KUKA KRL program: EPS_2_26115_SA7012_A_20260219035554.src

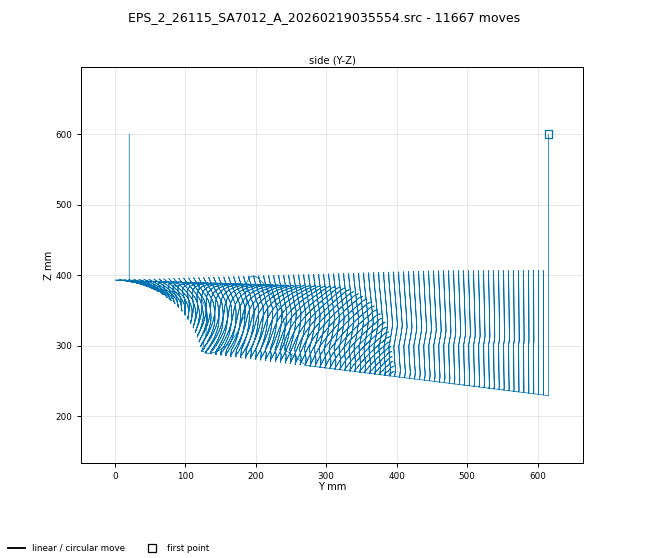
[picture p0: tool path of EPS_2_26115_SA7012_A_20260219035554.src, 11667 of 11669 moves have a stored position in this frame; points joined in program order, loops and branches not executed]
&ACCESS RVP
&REL 4
&COMMENT QRS 19112012
&PARAM EDITMASK = *
DEF PART()
EXT BAS (BAS_COMMAND :IN,REAL :IN )
INT I
BAS (#INITMOV,0 )

;KUKA QRS Post kuka4.cps  Date:22-06-2017 !

File_ID=3068

QRS_PRE_INIT()

;Init var - Until changes are made in qrs_pre_init
Outlet_Square_prg=0
Inlet_1_Square_prg=0
Inlet_2_Square_prg=0
Inlet_3_Square_prg=0
Inlet_4_Square_prg=0
Inlet_5_Square_prg=0

Outlet_1={X 0.000, Y 460.000, Z 306.500, B 0.000, E1 0.000 }
Inlet_1={X 0.000, Y 560.070, Z 281.500, B 0.000, E1 180.000 }
Outlet_1_type=201
Inlet_1_type=0
;QRS#1=Sidecore dimensions
;QRS#2=200-8" PVC SDR 35 Cut Back
;QRS#3=DeadEnd 201
;QRS#4=
;QRS#5=
;QRS#6=
;QRS#7=
;QRS#8=
;QRS#9=12-08 PSX
;QRS#10=

;QRS#11=
;QRS#12=
;QRS#13=
;QRS#14=
;QRS#15=
;QRS#16=1220x127x686 2,25'
;QRS#17=EPS Height
;QRS#18=407
;QRS#19=*
;QRS#20= UPDATED VERSION 22-06-2017
;QRS#21=*
Outlet_Square=0100
Inlet_1_Square=00
Inlet_2_Square=0
Inlet_3_Square=0
Inlet_4_Square=0
Inlet_5_Square=0
Mill_Square=1
Outlet_Square_Prg=214
Inlet_1_Square_prg=0

QRS_INIT()

$ADVANCE=5

; T1
PTP {E1 173.647,E2 173.647}
PTP {X 0,Y 615.427,A -85,B 0,C 180,E1 173.647,E2 173.647,E3 0,E4 0,E5 0,E6 0}
QRS_SPEED_INIT()
LIN {X 0,Y 615.427,Z 600,A -85,B 0,C 180,E1 173.647,E2 173.647,E3 0,E4 0,E5 0,E6 0} C_VEL
LIN {X 0,Y 615.427,Z 239.376,A -85,B 0,C 180,E1 173.647,E2 173.647} C_VEL
LIN {X 0,Y 615.427,Z 231.196,A -85,B 0,C 180,E1 173.647,E2 173.647} C_VEL
LIN {X 0,Y 615.428,Z 229.196,A -85,B 0,C 180,E1 173.461,E2 173.461} C_VEL
LIN {X 0,Y 615.493,Z 229.194,A -85,B 0,C 180,E1 170.806,E2 170.806} C_VEL
LIN {X 0,Y 615.44,Z 229.198,A -85,B 0,C 180,E1 168.143,E2 168.143} C_VEL
LIN {X 0,Y 615.432,Z 229.198,A -85,B 0,C 180,E1 166.084,E2 166.084} C_VEL
LIN {X 0,Y 615.43,Z 229.198,A -85,B 0,C 180,E1 164.098,E2 164.098} C_VEL
LIN {X 0,Y 615.426,Z 229.198,A -85,B 0,C 180,E1 162.046,E2 162.046} C_VEL
LIN {X 0,Y 615.472,Z 229.195,A -85,B 0,C 180,E1 159.274,E2 159.274} C_VEL
LIN {X 0,Y 615.435,Z 229.198,A -85,B 0,C 180,E1 156.447,E2 156.447} C_VEL
LIN {X 0,Y 615.425,Z 229.198,A -85,B 0,C 180,E1 154.287,E2 154.287} C_VEL
LIN {X 0,Y 615.424,Z 229.197,A -85,B 0,C 180,E1 152.088,E2 152.088} C_VEL
LIN {X 0,Y 615.437,Z 229.197,A -85,B 0,C 180,E1 149.844,E2 149.844} C_VEL
LIN {X 0,Y 615.473,Z 229.197,A -85,B 0,C 180,E1 147.548,E2 147.548} C_VEL
LIN {X 0,Y 615.476,Z 229.2,A -85,B 0,C 180,E1 145.191,E2 145.191} C_VEL
LIN {X 0,Y 615.429,Z 229.199,A -85,B 0,C 180,E1 142.761,E2 142.761} C_VEL
LIN {X 0,Y 615.456,Z 229.197,A -85,B 0,C 180,E1 139.913,E2 139.913} C_VEL
LIN {X 0,Y 615.499,Z 229.197,A -85,B 0,C 180,E1 137.656,E2 137.656} C_VEL
LIN {X 0,Y 615.424,Z 229.199,A -85,B 0,C 180,E1 134.934,E2 134.934} C_VEL
LIN {X 0,Y 615.463,Z 229.197,A -85,B 0,C 180,E1 132.087,E2 132.087} C_VEL
LIN {X 0,Y 615.485,Z 229.201,A -85,B 0,C 180,E1 129.749,E2 129.749} C_VEL
LIN {X 0,Y 615.428,Z 229.199,A -85,B 0,C 180,E1 127.246,E2 127.246} C_VEL
LIN {X 0,Y 615.421,Z 229.198,A -85,B 0,C 180,E1 124.819,E2 124.819} C_VEL
LIN {X 0,Y 615.465,Z 229.198,A -85,B 0,C 180,E1 122.34,E2 122.34} C_VEL
LIN {X 0,Y 615.456,Z 229.2,A -85,B 0,C 180,E1 119.803,E2 119.803} C_VEL
LIN {X 0,Y 615.416,Z 229.199,A -85,B 0,C 180,E1 117.18,E2 117.18} C_VEL
LIN {X 0,Y 615.483,Z 229.204,A -85,B 0,C 180,E1 114.272,E2 114.272} C_VEL
LIN {X 0,Y 615.466,Z 229.201,A -85,B 0,C 180,E1 112.137,E2 112.137} C_VEL
LIN {X 0,Y 615.449,Z 229.2,A -85,B 0,C 180,E1 110.034,E2 110.034} C_VEL
LIN {X 0,Y 615.435,Z 229.2,A -85,B 0,C 180,E1 107.958,E2 107.958} C_VEL
LIN {X 0,Y 615.427,Z 229.2,A -85,B 0,C 180,E1 105.906,E2 105.906} C_VEL
LIN {X 0,Y 615.421,Z 229.2,A -85,B 0,C 180,E1 103.875,E2 103.875} C_VEL
LIN {X 0,Y 615.418,Z 229.2,A -85,B 0,C 180,E1 101.862,E2 101.862} C_VEL
LIN {X 0,Y 615.416,Z 229.2,A -85,B 0,C 180,E1 99.863,E2 99.863} C_VEL
LIN {X 0,Y 615.413,Z 229.2,A -85,B 0,C 180,E1 97.876,E2 97.876} C_VEL
LIN {X 0,Y 615.413,Z 229.2,A -85,B 0,C 180,E1 95.899,E2 95.899} C_VEL
LIN {X 0,Y 615.448,Z 229.2,A -85,B 0,C 180,E1 93.273,E2 93.273} C_VEL
LIN {X 0,Y 615.453,Z 229.2,A -85,B 0,C 180,E1 90.654,E2 90.654} C_VEL
LIN {X 0,Y 615.413,Z 229.2,A -85,B 0,C 180,E1 88.037,E2 88.037} C_VEL
LIN {X 0,Y 615.459,Z 229.2,A -85,B 0,C 180,E1 85.415,E2 85.415} C_VEL
LIN {X 0,Y 615.44,Z 229.2,A -85,B 0,C 180,E1 82.784,E2 82.784} C_VEL
LIN {X 0,Y 615.439,Z 229.199,A -85,B 0,C 180,E1 80.801,E2 80.801} C_VEL
LIN {X 0,Y 615.435,Z 229.199,A -85,B 0,C 180,E1 78.806,E2 78.806} C_VEL
LIN {X 0,Y 615.43,Z 229.199,A -85,B 0,C 180,E1 76.798,E2 76.798} C_VEL
LIN {X 0,Y 615.425,Z 229.199,A -85,B 0,C 180,E1 74.773,E2 74.773} C_VEL
LIN {X 0,Y 615.42,Z 229.199,A -85,B 0,C 180,E1 72.728,E2 72.728} C_VEL
LIN {X 0,Y 615.417,Z 229.199,A -85,B 0,C 180,E1 70.66,E2 70.66} C_VEL
LIN {X 0,Y 615.416,Z 229.199,A -85,B 0,C 180,E1 68.566,E2 68.566} C_VEL
LIN {X 0,Y 615.461,Z 229.2,A -85,B 0,C 180,E1 65.98,E2 65.98} C_VEL
LIN {X 0,Y 615.471,Z 229.198,A -85,B 0,C 180,E1 63.556,E2 63.556} C_VEL
LIN {X 0,Y 615.441,Z 229.198,A -85,B 0,C 180,E1 61.34,E2 61.34} C_VEL
LIN {X 0,Y 615.42,Z 229.199,A -85,B 0,C 180,E1 59.077,E2 59.077} C_VEL
LIN {X 0,Y 615.441,Z 229.199,A -85,B 0,C 180,E1 56.46,E2 56.46} C_VEL
LIN {X 0,Y 615.443,Z 229.198,A -85,B 0,C 180,E1 53.573,E2 53.573} C_VEL
LIN {X 0,Y 615.422,Z 229.199,A -85,B 0,C 180,E1 50.935,E2 50.935} C_VEL
LIN {X 0,Y 615.459,Z 229.2,A -85,B 0,C 180,E1 48.525,E2 48.525} C_VEL
LIN {X 0,Y 615.446,Z 229.198,A -85,B 0,C 180,E1 45.848,E2 45.848} C_VEL
LIN {X 0,Y 615.421,Z 229.198,A -85,B 0,C 180,E1 43.242,E2 43.242} C_VEL
LIN {X 0,Y 615.428,Z 229.199,A -85,B 0,C 180,E1 41.089,E2 41.089} C_VEL
LIN {X 0,Y 615.45,Z 229.199,A -85,B 0,C 180,E1 38.899,E2 38.899} C_VEL
LIN {X 0,Y 615.473,Z 229.2,A -85,B 0,C 180,E1 36.418,E2 36.418} C_VEL
LIN {X 0,Y 615.437,Z 229.197,A -85,B 0,C 180,E1 34.018,E2 34.018} C_VEL
LIN {X 0,Y 615.42,Z 229.198,A -85,B 0,C 180,E1 31.683,E2 31.683} C_VEL
LIN {X 0,Y 615.433,Z 229.199,A -85,B 0,C 180,E1 29.403,E2 29.403} C_VEL
LIN {X 0,Y 615.476,Z 229.2,A -85,B 0,C 180,E1 27.045,E2 27.045} C_VEL
LIN {X 0,Y 615.436,Z 229.197,A -85,B 0,C 180,E1 24.268,E2 24.268} C_VEL
LIN {X 0,Y 615.427,Z 229.197,A -85,B 0,C 180,E1 22.133,E2 22.133} C_VEL
LIN {X 0,Y 615.424,Z 229.197,A -85,B 0,C 180,E1 20.03,E2 20.03} C_VEL
LIN {X 0,Y 615.481,Z 229.201,A -85,B 0,C 180,E1 17.266,E2 17.266} C_VEL
LIN {X 0,Y 615.436,Z 229.196,A -85,B 0,C 180,E1 14.545,E2 14.545} C_VEL
LIN {X 0,Y 615.433,Z 229.196,A -85,B 0,C 180,E1 12.527,E2 12.527} C_VEL
LIN {X 0,Y 615.431,Z 229.196,A -85,B 0,C 180,E1 10.523,E2 10.523} C_VEL
LIN {X 0,Y 615.428,Z 229.197,A -85,B 0,C 180,E1 8.533,E2 8.533} C_VEL
LIN {X 0,Y 615.428,Z 229.196,A -85,B 0,C 180,E1 6.539,E2 6.539} C_VEL
LIN {X 0,Y 615.428,Z 229.196,A -85,B 0,C 180,E1 4.581,E2 4.581} C_VEL
LIN {X 0,Y 615.457,Z 229.199,A -85,B 0,C 180,E1 1.959,E2 1.959} C_VEL
LIN {X 0,Y 615.473,Z 229.194,A -85,B 0,C 180,E1 -0.658,E2 -0.658} C_VEL
LIN {X 0,Y 615.428,Z 229.196,A -85,B 0,C 180,E1 -3.277,E2 -3.277} C_VEL
LIN {X 0,Y 615.467,Z 229.199,A -85,B 0,C 180,E1 -5.902,E2 -5.902} C_VEL
LIN {X 0,Y 615.463,Z 229.194,A -85,B 0,C 180,E1 -8.54,E2 -8.54} C_VEL
LIN {X 0,Y 615.43,Z 229.197,A -85,B 0,C 180,E1 -11.197,E2 -11.197} C_VEL
LIN {X 0,Y 615.499,Z 229.199,A -85,B 0,C 180,E1 -13.941,E2 -13.941} C_VEL
LIN {X 0,Y 615.438,Z 229.195,A -85,B 0,C 180,E1 -16.591,E2 -16.591} C_VEL
LIN {X 0,Y 615.435,Z 229.195,A -85,B 0,C 180,E1 -18.65,E2 -18.65} C_VEL
LIN {X 0,Y 615.432,Z 229.196,A -85,B 0,C 180,E1 -20.735,E2 -20.735} C_VEL
LIN {X 0,Y 615.481,Z 229.202,A -85,B 0,C 180,E1 -23.559,E2 -23.559} C_VEL
LIN {X 0,Y 615.499,Z 229.194,A -85,B 0,C 180,E1 -25.718,E2 -25.718} C_VEL
LIN {X 0,Y 615.43,Z 229.197,A -85,B 0,C 180,E1 -28.663,E2 -28.663} C_VEL
LIN {X 0,Y 615.462,Z 229.199,A -85,B 0,C 180,E1 -31.084,E2 -31.084} C_VEL
LIN {X 0,Y 615.447,Z 229.194,A -85,B 0,C 180,E1 -34.027,E2 -34.027} C_VEL
LIN {X 0,Y 615.434,Z 229.196,A -85,B 0,C 180,E1 -36.431,E2 -36.431} C_VEL
LIN {X 0,Y 615.488,Z 229.2,A -85,B 0,C 180,E1 -39.063,E2 -39.063} C_VEL
LIN {X 0,Y 615.482,Z 229.191,A -85,B 0,C 180,E1 -41.476,E2 -41.476} C_VEL
LIN {X 0,Y 615.435,Z 229.195,A -85,B 0,C 180,E1 -44.156,E2 -44.156} C_VEL
LIN {X 0,Y 615.478,Z 229.199,A -85,B 0,C 180,E1 -46.756,E2 -46.756} C_VEL
LIN {X 0,Y 615.478,Z 229.338,A -85,B 0,C 180,E1 -48.716,E2 -48.716} C_VEL
LIN {X 0,Y 615.493,Z 234.318,A -85,B 0,C 180,E1 -51.097,E2 -51.097} C_VEL
LIN {X 0,Y 615.453,Z 239.696,A -85,B 0,C 180,E1 -53.574,E2 -53.574} C_VEL
LIN {X 0,Y 615.494,Z 246.171,A -85,B 0,C 180,E1 -56.467,E2 -56.467} C_VEL
LIN {X 0,Y 615.478,Z 252.224,A -85,B 0,C 180,E1 -59.08,E2 -59.08} C_VEL
LIN {X 0,Y 615.475,Z 258.104,A -85,B 0,C 180,E1 -61.553,E2 -61.553} C_VEL
LIN {X 0,Y 615.479,Z 264.742,A -85,B 0,C 180,E1 -64.284,E2 -64.284} C_VEL
LIN {X 0,Y 615.484,Z 270.106,A -85,B 0,C 180,E1 -66.444,E2 -66.444} C_VEL
LIN {X 0,Y 615.489,Z 277.253,A -85,B 0,C 180,E1 -69.27,E2 -69.27} C_VEL
LIN {X 0,Y 615.465,Z 284.402,A -85,B 0,C 180,E1 -72.043,E2 -72.043} C_VEL
LIN {X 0,Y 615.495,Z 291.538,A -85,B 0,C 180,E1 -74.774,E2 -74.774} C_VEL
LIN {X 0,Y 615.442,Z 298.683,A -85,B 0,C 180,E1 -77.469,E2 -77.469} C_VEL
LIN {X 0,Y 615.497,Z 301.074,A -85,B 0,C 180,E1 -78.369,E2 -78.369} C_VEL
LIN {X 0,Y 615.482,Z 316.869,A -85,B 0,C 180,E1 -78.724,E2 -78.724} C_VEL
LIN {X 0,Y 615.443,Z 329.251,A -85,B 0,C 180,E1 -79.136,E2 -79.136} C_VEL
LIN {X 0,Y 615.439,Z 340.489,A -85,B 0,C 180,E1 -79.639,E2 -79.639} C_VEL
LIN {X 0,Y 615.489,Z 351.997,A -85,B 0,C 180,E1 -80.304,E2 -80.304} C_VEL
LIN {X 0,Y 615.499,Z 362.343,A -85,B 0,C 180,E1 -81.05,E2 -81.05} C_VEL
LIN {X 0,Y 615.497,Z 370.813,A -85,B 0,C 180,E1 -81.794,E2 -81.794} C_VEL
LIN {X 0,Y 615.498,Z 378.607,A -85,B 0,C 180,E1 -82.62,E2 -82.62} C_VEL
LIN {X 0,Y 615.496,Z 386.204,A -85,B 0,C 180,E1 -83.608,E2 -83.608} C_VEL
LIN {X 0,Y 615.498,Z 393.205,A -85,B 0,C 180,E1 -84.759,E2 -84.759} C_VEL
LIN {X 0,Y 615.493,Z 397.852,A -85,B 0,C 180,E1 -85.744,E2 -85.744} C_VEL
LIN {X 0,Y 615.494,Z 401.399,A -85,B 0,C 180,E1 -86.727,E2 -86.727} C_VEL
LIN {X 0,Y 615.497,Z 403.233,A -85,B 0,C 180,E1 -87.382,E2 -87.382} C_VEL
LIN {X 0,Y 615.5,Z 404.608,A -85,B 0,C 180,E1 -88.037,E2 -88.037} C_VEL
LIN {X 0,Y 615.496,Z 406.173,A -85,B 0,C 180,E1 -89.346,E2 -89.346} C_VEL
LIN {X 0,Y 615.494,Z 406.389,A -85,B 0,C 180,E1 -90,E2 -90} C_VEL
LIN {X 0,Y 615.495,Z 405.58,A -85,B 0,C 180,E1 -91.309,E2 -91.309} C_VEL
LIN {X 0,Y 615.5,Z 404.608,A -85,B 0,C 180,E1 -91.963,E2 -91.963} C_VEL
LIN {X 0,Y 615.497,Z 403.233,A -85,B 0,C 180,E1 -92.618,E2 -92.618} C_VEL
LIN {X 0,Y 615.496,Z 400.35,A -85,B 0,C 180,E1 -93.601,E2 -93.601} C_VEL
LIN {X 0,Y 615.498,Z 396.442,A -85,B 0,C 180,E1 -94.584,E2 -94.584} C_VEL
LIN {X 0,Y 615.499,Z 391.405,A -85,B 0,C 180,E1 -95.57,E2 -95.57} C_VEL
LIN {X 0,Y 615.497,Z 384.875,A -85,B 0,C 180,E1 -96.583,E2 -96.583} C_VEL
LIN {X 0,Y 615.497,Z 377.134,A -85,B 0,C 180,E1 -97.545,E2 -97.545} C_VEL
LIN {X 0,Y 615.498,Z 369.047,A -85,B 0,C 180,E1 -98.371,E2 -98.371} C_VEL
LIN {X 0,Y 615.499,Z 359.17,A -85,B 0,C 180,E1 -99.198,E2 -99.198} C_VEL
LIN {X 0,Y 615.471,Z 347.987,A -85,B 0,C 180,E1 -99.945,E2 -99.945} C_VEL
LIN {X 0,Y 615.435,Z 337.035,A -85,B 0,C 180,E1 -100.528,E2 -100.528} C_VEL
LIN {X 0,Y 615.454,Z 324.825,A -85,B 0,C 180,E1 -101.029,E2 -101.029} C_VEL
LIN {X 0,Y 615.495,Z 312.073,A -85,B 0,C 180,E1 -101.401,E2 -101.401} C_VEL
LIN {X 0,Y 615.497,Z 301.074,A -85,B 0,C 180,E1 -101.631,E2 -101.631} C_VEL
LIN {X 0,Y 615.467,Z 294.99,A -85,B 0,C 180,E1 -103.923,E2 -103.923} C_VEL
LIN {X 0,Y 615.463,Z 287.97,A -85,B 0,C 180,E1 -106.587,E2 -106.587} C_VEL
LIN {X 0,Y 615.487,Z 280.835,A -85,B 0,C 180,E1 -109.338,E2 -109.338} C_VEL
LIN {X 0,Y 615.474,Z 273.68,A -85,B 0,C 180,E1 -112.137,E2 -112.137} C_VEL
LIN {X 0,Y 615.483,Z 266.537,A -85,B 0,C 180,E1 -114.991,E2 -114.991} C_VEL
LIN {X 0,Y 615.489,Z 259.377,A -85,B 0,C 180,E1 -117.914,E2 -117.914} C_VEL
LIN {X 0,Y 615.48,Z 254.015,A -85,B 0,C 180,E1 -120.16,E2 -120.16} C_VEL
LIN {X 0,Y 615.461,Z 248.65,A -85,B 0,C 180,E1 -122.458,E2 -122.458} C_VEL
LIN {X 0,Y 615.476,Z 243.274,A -85,B 0,C 180,E1 -124.815,E2 -124.815} C_VEL
LIN {X 0,Y 615.491,Z 237.901,A -85,B 0,C 180,E1 -127.241,E2 -127.241} C_VEL
LIN {X 0,Y 615.443,Z 232.534,A -85,B 0,C 180,E1 -129.753,E2 -129.753} C_VEL
LIN {X 0,Y 615.469,Z 229.199,A -85,B 0,C 180,E1 -131.379,E2 -131.379} C_VEL
LIN {X 0,Y 615.436,Z 229.195,A -85,B 0,C 180,E1 -133.991,E2 -133.991} C_VEL
LIN {X 0,Y 615.437,Z 229.195,A -85,B 0,C 180,E1 -136.006,E2 -136.006} C_VEL
LIN {X 0,Y 615.478,Z 229.192,A -85,B 0,C 180,E1 -138.523,E2 -138.523} C_VEL
LIN {X 0,Y 615.468,Z 229.199,A -85,B 0,C 180,E1 -141.092,E2 -141.092} C_VEL
LIN {X 0,Y 615.434,Z 229.196,A -85,B 0,C 180,E1 -143.569,E2 -143.569} C_VEL
LIN {X 0,Y 615.496,Z 229.193,A -85,B 0,C 180,E1 -146.463,E2 -146.463} C_VEL
LIN {X 0,Y 615.447,Z 229.198,A -85,B 0,C 180,E1 -149.076,E2 -149.076} C_VEL
LIN {X 0,Y 615.432,Z 229.196,A -85,B 0,C 180,E1 -151.557,E2 -151.557} C_VEL
LIN {X 0,Y 615.5,Z 229.199,A -85,B 0,C 180,E1 -154.427,E2 -154.427} C_VEL
LIN {X 0,Y 615.432,Z 229.196,A -85,B 0,C 180,E1 -157.151,E2 -157.151} C_VEL
LIN {X 0,Y 615.479,Z 229.194,A -85,B 0,C 180,E1 -159.964,E2 -159.964} C_VEL
LIN {X 0,Y 615.441,Z 229.198,A -85,B 0,C 180,E1 -162.725,E2 -162.725} C_VEL
LIN {X 0,Y 615.436,Z 229.197,A -85,B 0,C 180,E1 -164.77,E2 -164.77} C_VEL
LIN {X 0,Y 615.433,Z 229.197,A -85,B 0,C 180,E1 -166.794,E2 -166.794} C_VEL
LIN {X 0,Y 615.434,Z 229.195,A -85,B 0,C 180,E1 -169.132,E2 -169.132} C_VEL
LIN {X 0,Y 615.463,Z 229.194,A -85,B 0,C 180,E1 -171.46,E2 -171.46} C_VEL
LIN {X 0,Y 615.467,Z 229.199,A -85,B 0,C 180,E1 -174.098,E2 -174.098} C_VEL
LIN {X 0,Y 615.428,Z 229.196,A -85,B 0,C 180,E1 -176.723,E2 -176.723} C_VEL
LIN {X 0,Y 615.47,Z 229.195,A -85,B 0,C 180,E1 -179.342,E2 -179.342} C_VEL
LIN {X 0,Y 615.457,Z 229.199,A -85,B 0,C 180,E1 -181.959,E2 -181.959} C_VEL
LIN {X 0,Y 615.428,Z 229.196,A -85,B 0,C 180,E1 -184.581,E2 -184.581} C_VEL
LIN {X 0,Y 615.428,Z 229.196,A -85,B 0,C 180,E1 -186.539,E2 -186.539} C_VEL
LIN {X 0,Y 614.793,Z 229.344,A -85,B 0,C 180,E1 -187.085,E2 -187.085} C_VEL
LIN {X 0,Y 611.998,Z 229.748,A -85,B 0,C 180,E1 -187.971,E2 -187.971} C_VEL
LIN {X 0,Y 609.607,Z 230.064,A -85,B 0,C 180,E1 -188.684,E2 -188.684} C_VEL
LIN {X 0,Y 608.552,Z 230.185,A -85,B 0,C 180,E1 -189.234,E2 -189.234} C_VEL
LIN {X 0,Y 608.451,Z 230.194,A -85,B 0,C 180,E1 -189.42,E2 -189.42} C_VEL
LIN {X 0,Y 608.418,Z 230.193,A -85,B 0,C 180,E1 -191.996,E2 -191.996} C_VEL
LIN {X 0,Y 608.399,Z 230.195,A -85,B 0,C 180,E1 -194.034,E2 -194.034} C_VEL
LIN {X 0,Y 608.429,Z 230.192,A -85,B 0,C 180,E1 -196.52,E2 -196.52} C_VEL
LIN {X 0,Y 608.419,Z 230.195,A -85,B 0,C 180,E1 -199.566,E2 -199.566} C_VEL
LIN {X 0,Y 608.429,Z 230.192,A -85,B 0,C 180,E1 -202.401,E2 -202.401} C_VEL
LIN {X 0,Y 608.421,Z 230.196,A -85,B 0,C 180,E1 -205.296,E2 -205.296} C_VEL
LIN {X 0,Y 608.408,Z 230.194,A -85,B 0,C 180,E1 -207.514,E2 -207.514} C_VEL
LIN {X 0,Y 608.411,Z 230.193,A -85,B 0,C 180,E1 -209.964,E2 -209.964} C_VEL
LIN {X 0,Y 608.423,Z 230.199,A -85,B 0,C 180,E1 -212.875,E2 -212.875} C_VEL
LIN {X 0,Y 608.401,Z 230.195,A -85,B 0,C 180,E1 -215.273,E2 -215.273} C_VEL
LIN {X 0,Y 608.423,Z 230.192,A -85,B 0,C 180,E1 -217.742,E2 -217.742} C_VEL
LIN {X 0,Y 608.435,Z 230.198,A -85,B 0,C 180,E1 -220.328,E2 -220.328} C_VEL
LIN {X 0,Y 608.404,Z 230.196,A -85,B 0,C 180,E1 -222.956,E2 -222.956} C_VEL
LIN {X 0,Y 608.396,Z 230.195,A -85,B 0,C 180,E1 -225.2,E2 -225.2} C_VEL
LIN {X 0,Y 608.44,Z 230.194,A -85,B 0,C 180,E1 -227.938,E2 -227.938} C_VEL
LIN {X 0,Y 608.426,Z 230.193,A -85,B 0,C 180,E1 -230.697,E2 -230.697} C_VEL
LIN {X 0,Y 608.39,Z 230.195,A -85,B 0,C 180,E1 -233.081,E2 -233.081} C_VEL
LIN {X 0,Y 608.428,Z 230.193,A -85,B 0,C 180,E1 -235.529,E2 -235.529} C_VEL
LIN {X 0,Y 608.437,Z 230.199,A -85,B 0,C 180,E1 -237.905,E2 -237.905} C_VEL
LIN {X 0,Y 608.438,Z 230.194,A -85,B 0,C 180,E1 -240.219,E2 -240.219} C_VEL
LIN {X 0,Y 608.411,Z 230.193,A -85,B 0,C 180,E1 -242.79,E2 -242.79} C_VEL
LIN {X 0,Y 608.453,Z 230.196,A -85,B 0,C 180,E1 -245.836,E2 -245.836} C_VEL
LIN {X 0,Y 608.417,Z 230.193,A -85,B 0,C 180,E1 -248.307,E2 -248.307} C_VEL
LIN {X 0,Y 608.431,Z 230.194,A -85,B 0,C 180,E1 -251.13,E2 -251.13} C_VEL
LIN {X 0,Y 608.417,Z 230.196,A -85,B 0,C 180,E1 -253.905,E2 -253.905} C_VEL
LIN {X 0,Y 608.402,Z 230.196,A -85,B 0,C 180,E1 -255.978,E2 -255.978} C_VEL
LIN {X 0,Y 608.406,Z 230.195,A -85,B 0,C 180,E1 -257.999,E2 -257.999} C_VEL
LIN {X 0,Y 608.395,Z 230.196,A -85,B 0,C 180,E1 -260.022,E2 -260.022} C_VEL
LIN {X 0,Y 608.411,Z 230.193,A -85,B 0,C 180,E1 -262.032,E2 -262.032} C_VEL
LIN {X 0,Y 608.42,Z 230.195,A -85,B 0,C 180,E1 -264.698,E2 -264.698} C_VEL
LIN {X 0,Y 608.442,Z 230.195,A -85,B 0,C 180,E1 -267.352,E2 -267.352} C_VEL
LIN {X 0,Y 608.403,Z 230.194,A -85,B 0,C 180,E1 -270,E2 -270} C_VEL
LIN {X 0,Y 608.442,Z 230.195,A -85,B 0,C 180,E1 -272.648,E2 -272.648} C_VEL
LIN {X 0,Y 608.42,Z 230.195,A -85,B 0,C 180,E1 -275.302,E2 -275.302} C_VEL
LIN {X 0,Y 608.411,Z 230.193,A -85,B 0,C 180,E1 -277.968,E2 -277.968} C_VEL
LIN {X 0,Y 608.444,Z 230.199,A -85,B 0,C 180,E1 -280.65,E2 -280.65} C_VEL
LIN {X 0,Y 608.405,Z 230.194,A -85,B 0,C 180,E1 -283.357,E2 -283.357} C_VEL
LIN {X 0,Y 608.409,Z 230.193,A -85,B 0,C 180,E1 -285.407,E2 -285.407} C_VEL
LIN {X 0,Y 608.39,Z 230.195,A -85,B 0,C 180,E1 -287.478,E2 -287.478} C_VEL
LIN {X 0,Y 608.393,Z 230.195,A -85,B 0,C 180,E1 -289.572,E2 -289.572} C_VEL
LIN {X 0,Y 608.476,Z 230.194,A -85,B 0,C 180,E1 -292.405,E2 -292.405} C_VEL
LIN {X 0,Y 608.418,Z 230.197,A -85,B 0,C 180,E1 -294.572,E2 -294.572} C_VEL
LIN {X 0,Y 608.411,Z 230.193,A -85,B 0,C 180,E1 -297.21,E2 -297.21} C_VEL
LIN {X 0,Y 608.468,Z 230.194,A -85,B 0,C 180,E1 -299.985,E2 -299.985} C_VEL
LIN {X 0,Y 608.404,Z 230.194,A -85,B 0,C 180,E1 -302.882,E2 -302.882} C_VEL
LIN {X 0,Y 608.397,Z 230.196,A -85,B 0,C 180,E1 -305.28,E2 -305.28} C_VEL
LIN {X 0,Y 608.438,Z 230.194,A -85,B 0,C 180,E1 -308.247,E2 -308.247} C_VEL
LIN {X 0,Y 608.426,Z 230.193,A -85,B 0,C 180,E1 -310.336,E2 -310.336} C_VEL
LIN {X 0,Y 608.395,Z 230.195,A -85,B 0,C 180,E1 -312.964,E2 -312.964} C_VEL
LIN {X 0,Y 608.439,Z 230.198,A -85,B 0,C 180,E1 -315.737,E2 -315.737} C_VEL
LIN {X 0,Y 608.437,Z 230.194,A -85,B 0,C 180,E1 -317.945,E2 -317.945} C_VEL
LIN {X 0,Y 608.395,Z 230.195,A -85,B 0,C 180,E1 -320.71,E2 -320.71} C_VEL
LIN {X 0,Y 608.424,Z 230.196,A -85,B 0,C 180,E1 -323.09,E2 -323.09} C_VEL
LIN {X 0,Y 608.452,Z 230.195,A -85,B 0,C 180,E1 -325.537,E2 -325.537} C_VEL
LIN {X 0,Y 608.425,Z 230.192,A -85,B 0,C 180,E1 -327.91,E2 -327.91} C_VEL
LIN {X 0,Y 608.409,Z 230.193,A -85,B 0,C 180,E1 -330.224,E2 -330.224} C_VEL
LIN {X 0,Y 608.454,Z 230.192,A -85,B 0,C 180,E1 -332.795,E2 -332.795} C_VEL
LIN {X 0,Y 608.425,Z 230.191,A -85,B 0,C 180,E1 -335.856,E2 -335.856} C_VEL
LIN {X 0,Y 608.425,Z 230.192,A -85,B 0,C 180,E1 -338.312,E2 -338.312} C_VEL
LIN {X 0,Y 608.441,Z 230.193,A -85,B 0,C 180,E1 -341.289,E2 -341.289} C_VEL
LIN {X 0,Y 608.408,Z 230.193,A -85,B 0,C 180,E1 -343.91,E2 -343.91} C_VEL
LIN {X 0,Y 608.458,Z 230.197,A -85,B 0,C 180,E1 -346.648,E2 -346.648} C_VEL
LIN {X 0,Y 608.42,Z 230.192,A -85,B 0,C 180,E1 -349.354,E2 -349.354} C_VEL
LIN {X 0,Y 608.412,Z 230.193,A -85,B 0,C 180,E1 -351.368,E2 -351.368} C_VEL
LIN {X 0,Y 608.424,Z 230.194,A -85,B 0,C 180,E1 -354.037,E2 -354.037} C_VEL
LIN {X 0,Y 608.467,Z 230.191,A -85,B 0,C 180,E1 -356.693,E2 -356.693} C_VEL
LIN {X 0,Y 608.407,Z 230.193,A -85,B 0,C 180,E1 -359.342,E2 -359.342} C_VEL
LIN {X 0,Y 608.416,Z 230.192,A -85,B 0,C 180,E1 -361.328,E2 -361.328} C_VEL
LIN {X 0,Y 608.4,Z 230.194,A -85,B 0,C 180,E1 -363.315,E2 -363.315} C_VEL
LIN {X 0,Y 608.442,Z 230.197,A -85,B 0,C 180,E1 -365.971,E2 -365.971} C_VEL
LIN {X 0,Y 608.43,Z 230.192,A -85,B 0,C 180,E1 -368.64,E2 -368.64} C_VEL
LIN {X 0,Y 608.414,Z 230.194,A -85,B 0,C 180,E1 -371.328,E2 -371.328} C_VEL
LIN {X 0,Y 608.468,Z 230.194,A -85,B 0,C 180,E1 -374.041,E2 -374.041} C_VEL
LIN {X 0,Y 608.412,Z 230.193,A -85,B 0,C 180,E1 -376.788,E2 -376.788} C_VEL
LIN {X 0,Y 608.431,Z 230.198,A -85,B 0,C 180,E1 -379.574,E2 -379.574} C_VEL
LIN {X 0,Y 608.43,Z 230.191,A -85,B 0,C 180,E1 -382.472,E2 -382.472} C_VEL
LIN {X 0,Y 608.418,Z 230.192,A -85,B 0,C 180,E1 -384.575,E2 -384.575} C_VEL
LIN {X 0,Y 608.405,Z 230.194,A -85,B 0,C 180,E1 -386.779,E2 -386.779} C_VEL
LIN {X 0,Y 608.465,Z 230.191,A -85,B 0,C 180,E1 -389.782,E2 -389.782} C_VEL
LIN {X 0,Y 608.416,Z 230.192,A -85,B 0,C 180,E1 -392.517,E2 -392.517} C_VEL
LIN {X 0,Y 608.418,Z 230.196,A -85,B 0,C 180,E1 -394.903,E2 -394.903} C_VEL
LIN {X 0,Y 608.445,Z 230.191,A -85,B 0,C 180,E1 -397.75,E2 -397.75} C_VEL
LIN {X 0,Y 608.406,Z 230.194,A -85,B 0,C 180,E1 -400.325,E2 -400.325} C_VEL
LIN {X 0,Y 608.449,Z 230.198,A -85,B 0,C 180,E1 -402.962,E2 -402.962} C_VEL
LIN {X 0,Y 608.42,Z 230.193,A -85,B 0,C 180,E1 -405.742,E2 -405.742} C_VEL
LIN {X 0,Y 608.455,Z 230.313,A -85,B 0,C 180,E1 -408.525,E2 -408.525} C_VEL
LIN {X 0,Y 608.474,Z 234.678,A -85,B 0,C 180,E1 -410.704,E2 -410.704} C_VEL
LIN {X 0,Y 608.473,Z 239.769,A -85,B 0,C 180,E1 -413.087,E2 -413.087} C_VEL
LIN {X 0,Y 608.453,Z 245.159,A -85,B 0,C 180,E1 -415.53,E2 -415.53} C_VEL
LIN {X 0,Y 608.454,Z 250.548,A -85,B 0,C 180,E1 -417.906,E2 -417.906} C_VEL
LIN {X 0,Y 608.476,Z 255.938,A -85,B 0,C 180,E1 -420.222,E2 -420.222} C_VEL
LIN {X 0,Y 608.459,Z 262.086,A -85,B 0,C 180,E1 -422.798,E2 -422.798} C_VEL
LIN {X 0,Y 608.454,Z 268.513,A -85,B 0,C 180,E1 -425.429,E2 -425.429} C_VEL
LIN {X 0,Y 608.445,Z 275.699,A -85,B 0,C 180,E1 -428.308,E2 -428.308} C_VEL
LIN {X 0,Y 608.432,Z 282.885,A -85,B 0,C 180,E1 -431.13,E2 -431.13} C_VEL
LIN {X 0,Y 608.422,Z 290.071,A -85,B 0,C 180,E1 -433.905,E2 -433.905} C_VEL
LIN {X 0,Y 608.429,Z 297.257,A -85,B 0,C 180,E1 -436.643,E2 -436.643} C_VEL
LIN {X 0,Y 608.459,Z 301.63,A -85,B 0,C 180,E1 -438.254,E2 -438.254} C_VEL
LIN {X 0,Y 608.544,Z 314.708,A -85,B 0,C 180,E1 -438.53,E2 -438.53} C_VEL
LIN {X 0,Y 608.473,Z 327.572,A -85,B 0,C 180,E1 -438.942,E2 -438.942} C_VEL
LIN {X 0,Y 608.465,Z 338.926,A -85,B 0,C 180,E1 -439.435,E2 -439.435} C_VEL
LIN {X 0,Y 608.471,Z 349.581,A -85,B 0,C 180,E1 -440.023,E2 -440.023} C_VEL
LIN {X 0,Y 608.483,Z 360.477,A -85,B 0,C 180,E1 -440.778,E2 -440.778} C_VEL
LIN {X 0,Y 608.475,Z 371.114,A -85,B 0,C 180,E1 -441.699,E2 -441.699} C_VEL
LIN {X 0,Y 608.471,Z 378.961,A -85,B 0,C 180,E1 -442.534,E2 -442.534} C_VEL
LIN {X 0,Y 608.461,Z 386.29,A -85,B 0,C 180,E1 -443.485,E2 -443.485} C_VEL
LIN {X 0,Y 608.451,Z 391.866,A -85,B 0,C 180,E1 -444.366,E2 -444.366} C_VEL
LIN {X 0,Y 608.432,Z 396.951,A -85,B 0,C 180,E1 -445.362,E2 -445.362} C_VEL
LIN {X 0,Y 608.449,Z 400.896,A -85,B 0,C 180,E1 -446.358,E2 -446.358} C_VEL
LIN {X 0,Y 608.425,Z 403.809,A -85,B 0,C 180,E1 -447.352,E2 -447.352} C_VEL
LIN {X 0,Y 608.445,Z 405.201,A -85,B 0,C 180,E1 -448.014,E2 -448.014} C_VEL
LIN {X 0,Y 608.439,Z 406.783,A -85,B 0,C 180,E1 -449.338,E2 -449.338} C_VEL
LIN {X 0,Y 608.434,Z 406.999,A -85,B 0,C 180,E1 -450,E2 -450} C_VEL
LIN {X 0,Y 608.448,Z 406.184,A -85,B 0,C 180,E1 -451.324,E2 -451.324} C_VEL
LIN {X 0,Y 608.445,Z 405.201,A -85,B 0,C 180,E1 -451.986,E2 -451.986} C_VEL
LIN {X 0,Y 608.425,Z 403.809,A -85,B 0,C 180,E1 -452.648,E2 -452.648} C_VEL
LIN {X 0,Y 608.449,Z 400.896,A -85,B 0,C 180,E1 -453.642,E2 -453.642} C_VEL
LIN {X 0,Y 608.432,Z 396.951,A -85,B 0,C 180,E1 -454.638,E2 -454.638} C_VEL
LIN {X 0,Y 608.438,Z 390.877,A -85,B 0,C 180,E1 -455.801,E2 -455.801} C_VEL
LIN {X 0,Y 608.463,Z 384.236,A -85,B 0,C 180,E1 -456.799,E2 -456.799} C_VEL
LIN {X 0,Y 608.456,Z 375.991,A -85,B 0,C 180,E1 -457.8,E2 -457.8} C_VEL
LIN {X 0,Y 608.472,Z 367.535,A -85,B 0,C 180,E1 -458.636,E2 -458.636} C_VEL
LIN {X 0,Y 608.48,Z 357.091,A -85,B 0,C 180,E1 -459.473,E2 -459.473} C_VEL
LIN {X 0,Y 608.481,Z 346.758,A -85,B 0,C 180,E1 -460.145,E2 -460.145} C_VEL
LIN {X 0,Y 608.46,Z 335.898,A -85,B 0,C 180,E1 -460.711,E2 -460.711} C_VEL
LIN {X 0,Y 608.49,Z 324.113,A -85,B 0,C 180,E1 -461.185,E2 -461.185} C_VEL
LIN {X 0,Y 608.55,Z 311.273,A -85,B 0,C 180,E1 -461.554,E2 -461.554} C_VEL
LIN {X 0,Y 608.435,Z 301.468,A -85,B 0,C 180,E1 -461.768,E2 -461.768} C_VEL
LIN {X 0,Y 608.426,Z 295.461,A -85,B 0,C 180,E1 -464.038,E2 -464.038} C_VEL
LIN {X 0,Y 608.42,Z 288.275,A -85,B 0,C 180,E1 -466.785,E2 -466.785} C_VEL
LIN {X 0,Y 608.447,Z 281.089,A -85,B 0,C 180,E1 -469.57,E2 -469.57} C_VEL
LIN {X 0,Y 608.445,Z 275.699,A -85,B 0,C 180,E1 -471.692,E2 -471.692} C_VEL
LIN {X 0,Y 608.454,Z 268.513,A -85,B 0,C 180,E1 -474.571,E2 -474.571} C_VEL
LIN {X 0,Y 608.459,Z 262.086,A -85,B 0,C 180,E1 -477.202,E2 -477.202} C_VEL
LIN {X 0,Y 608.469,Z 255.487,A -85,B 0,C 180,E1 -479.97,E2 -479.97} C_VEL
LIN {X 0,Y 608.442,Z 249.579,A -85,B 0,C 180,E1 -482.518,E2 -482.518} C_VEL
LIN {X 0,Y 608.471,Z 244.18,A -85,B 0,C 180,E1 -484.907,E2 -484.907} C_VEL
LIN {X 0,Y 608.444,Z 237.973,A -85,B 0,C 180,E1 -487.747,E2 -487.747} C_VEL
LIN {X 0,Y 608.44,Z 232.537,A -85,B 0,C 180,E1 -490.326,E2 -490.326} C_VEL
LIN {X 0,Y 608.455,Z 230.318,A -85,B 0,C 180,E1 -491.475,E2 -491.475} C_VEL
LIN {X 0,Y 608.431,Z 230.191,A -85,B 0,C 180,E1 -493.872,E2 -493.872} C_VEL
LIN {X 0,Y 608.482,Z 230.19,A -85,B 0,C 180,E1 -496.689,E2 -496.689} C_VEL
LIN {X 0,Y 608.454,Z 230.197,A -85,B 0,C 180,E1 -498.821,E2 -498.821} C_VEL
LIN {X 0,Y 608.413,Z 230.195,A -85,B 0,C 180,E1 -501.406,E2 -501.406} C_VEL
LIN {X 0,Y 608.435,Z 230.19,A -85,B 0,C 180,E1 -503.955,E2 -503.955} C_VEL
LIN {X 0,Y 608.449,Z 230.192,A -85,B 0,C 180,E1 -506.326,E2 -506.326} C_VEL
LIN {X 0,Y 608.442,Z 230.198,A -85,B 0,C 180,E1 -508.732,E2 -508.732} C_VEL
LIN {X 0,Y 608.427,Z 230.191,A -85,B 0,C 180,E1 -511.386,E2 -511.386} C_VEL
LIN {X 0,Y 608.483,Z 230.191,A -85,B 0,C 180,E1 -514.275,E2 -514.275} C_VEL
LIN {X 0,Y 608.421,Z 230.194,A -85,B 0,C 180,E1 -516.872,E2 -516.872} C_VEL
LIN {X 0,Y 608.428,Z 230.191,A -85,B 0,C 180,E1 -519.328,E2 -519.328} C_VEL
LIN {X 0,Y 608.438,Z 230.193,A -85,B 0,C 180,E1 -521.825,E2 -521.825} C_VEL
LIN {X 0,Y 608.439,Z 230.193,A -85,B 0,C 180,E1 -524.59,E2 -524.59} C_VEL
LIN {X 0,Y 608.427,Z 230.193,A -85,B 0,C 180,E1 -526.64,E2 -526.64} C_VEL
LIN {X 0,Y 608.429,Z 230.192,A -85,B 0,C 180,E1 -529.346,E2 -529.346} C_VEL
LIN {X 0,Y 608.464,Z 230.195,A -85,B 0,C 180,E1 -532.029,E2 -532.029} C_VEL
LIN {X 0,Y 608.414,Z 230.193,A -85,B 0,C 180,E1 -534.694,E2 -534.694} C_VEL
LIN {X 0,Y 608.462,Z 230.19,A -85,B 0,C 180,E1 -537.348,E2 -537.348} C_VEL
LIN {X 0,Y 608.452,Z 230.193,A -85,B 0,C 180,E1 -539.996,E2 -539.996} C_VEL
LIN {X 0,Y 608.425,Z 230.191,A -85,B 0,C 180,E1 -542.644,E2 -542.644} C_VEL
LIN {X 0,Y 608.459,Z 230.193,A -85,B 0,C 180,E1 -545.298,E2 -545.298} C_VEL
LIN {X 0,Y 608.409,Z 230.196,A -85,B 0,C 180,E1 -547.963,E2 -547.963} C_VEL
LIN {X 0,Y 608.451,Z 230.194,A -85,B 0,C 180,E1 -549.42,E2 -549.42} C_VEL
LIN {X 0,Y 607.745,Z 230.278,A -85,B 0,C 180,E1 -549.972,E2 -549.972} C_VEL
LIN {X 0,Y 604.876,Z 230.636,A -85,B 0,C 180,E1 -550.869,E2 -550.869} C_VEL
LIN {X 0,Y 602.479,Z 230.938,A -85,B 0,C 180,E1 -551.591,E2 -551.591} C_VEL
LIN {X 0,Y 601.455,Z 231.06,A -85,B 0,C 180,E1 -552.147,E2 -552.147} C_VEL
LIN {X 0,Y 601.373,Z 231.07,A -85,B 0,C 180,E1 -552.336,E2 -552.336} C_VEL
LIN {X 0,Y 601.385,Z 231.073,A -85,B 0,C 180,E1 -554.893,E2 -554.893} C_VEL
LIN {X 0,Y 601.391,Z 231.074,A -85,B 0,C 180,E1 -556.982,E2 -556.982} C_VEL
LIN {X 0,Y 601.37,Z 231.071,A -85,B 0,C 180,E1 -559.805,E2 -559.805} C_VEL
LIN {X 0,Y 601.387,Z 231.072,A -85,B 0,C 180,E1 -562.601,E2 -562.601} C_VEL
LIN {X 0,Y 601.374,Z 231.079,A -85,B 0,C 180,E1 -564.874,E2 -564.874} C_VEL
LIN {X 0,Y 601.383,Z 231.071,A -85,B 0,C 180,E1 -567.358,E2 -567.358} C_VEL
LIN {X 0,Y 601.376,Z 231.071,A -85,B 0,C 180,E1 -569.389,E2 -569.389} C_VEL
LIN {X 0,Y 601.362,Z 231.071,A -85,B 0,C 180,E1 -571.723,E2 -571.723} C_VEL
LIN {X 0,Y 601.388,Z 231.07,A -85,B 0,C 180,E1 -574.114,E2 -574.114} C_VEL
LIN {X 0,Y 601.377,Z 231.079,A -85,B 0,C 180,E1 -576.577,E2 -576.577} C_VEL
LIN {X 0,Y 601.366,Z 231.072,A -85,B 0,C 180,E1 -579.122,E2 -579.122} C_VEL
LIN {X 0,Y 601.382,Z 231.07,A -85,B 0,C 180,E1 -581.76,E2 -581.76} C_VEL
LIN {X 0,Y 601.373,Z 231.077,A -85,B 0,C 180,E1 -584.531,E2 -584.531} C_VEL
LIN {X 0,Y 601.358,Z 231.071,A -85,B 0,C 180,E1 -587.326,E2 -587.326} C_VEL
LIN {X 0,Y 601.372,Z 231.077,A -85,B 0,C 180,E1 -590.003,E2 -590.003} C_VEL
LIN {X 0,Y 601.38,Z 231.071,A -85,B 0,C 180,E1 -592.614,E2 -592.614} C_VEL
LIN {X 0,Y 601.374,Z 231.069,A -85,B 0,C 180,E1 -595.066,E2 -595.066} C_VEL
LIN {X 0,Y 601.388,Z 231.07,A -85,B 0,C 180,E1 -597.482,E2 -597.482} C_VEL
LIN {X 0,Y 601.434,Z 231.071,A -85,B 0,C 180,E1 -599.837,E2 -599.837} C_VEL
LIN {X 0,Y 601.388,Z 231.068,A -85,B 0,C 180,E1 -602.886,E2 -602.886} C_VEL
LIN {X 0,Y 601.428,Z 231.071,A -85,B 0,C 180,E1 -605.859,E2 -605.859} C_VEL
LIN {X 0,Y 601.383,Z 231.072,A -85,B 0,C 180,E1 -608.04,E2 -608.04} C_VEL
LIN {X 0,Y 601.357,Z 231.073,A -85,B 0,C 180,E1 -610.189,E2 -610.189} C_VEL
LIN {X 0,Y 601.38,Z 231.072,A -85,B 0,C 180,E1 -613.013,E2 -613.013} C_VEL
LIN {X 0,Y 601.356,Z 231.075,A -85,B 0,C 180,E1 -615.903,E2 -615.903} C_VEL
LIN {X 0,Y 601.367,Z 231.073,A -85,B 0,C 180,E1 -617.857,E2 -617.857} C_VEL
LIN {X 0,Y 601.363,Z 231.072,A -85,B 0,C 180,E1 -620.583,E2 -620.583} C_VEL
LIN {X 0,Y 601.422,Z 231.073,A -85,B 0,C 180,E1 -623.289,E2 -623.289} C_VEL
LIN {X 0,Y 601.34,Z 231.074,A -85,B 0,C 180,E1 -625.979,E2 -625.979} C_VEL
LIN {X 0,Y 601.355,Z 231.072,A -85,B 0,C 180,E1 -627.991,E2 -627.991} C_VEL
LIN {X 0,Y 601.41,Z 231.07,A -85,B 0,C 180,E1 -630.67,E2 -630.67} C_VEL
LIN {X 0,Y 601.386,Z 231.072,A -85,B 0,C 180,E1 -633.35,E2 -633.35} C_VEL
LIN {X 0,Y 601.349,Z 231.073,A -85,B 0,C 180,E1 -636.038,E2 -636.038} C_VEL
LIN {X 0,Y 601.415,Z 231.075,A -85,B 0,C 180,E1 -638.738,E2 -638.738} C_VEL
LIN {X 0,Y 601.372,Z 231.07,A -85,B 0,C 180,E1 -641.459,E2 -641.459} C_VEL
LIN {X 0,Y 601.355,Z 231.072,A -85,B 0,C 180,E1 -643.517,E2 -643.517} C_VEL
LIN {X 0,Y 601.409,Z 231.072,A -85,B 0,C 180,E1 -646.287,E2 -646.287} C_VEL
LIN {X 0,Y 601.373,Z 231.071,A -85,B 0,C 180,E1 -649.1,E2 -649.1} C_VEL
LIN {X 0,Y 601.353,Z 231.072,A -85,B 0,C 180,E1 -651.241,E2 -651.241} C_VEL
LIN {X 0,Y 601.369,Z 231.07,A -85,B 0,C 180,E1 -653.412,E2 -653.412} C_VEL
LIN {X 0,Y 601.366,Z 231.075,A -85,B 0,C 180,E1 -655.874,E2 -655.874} C_VEL
LIN {X 0,Y 601.391,Z 231.07,A -85,B 0,C 180,E1 -658.628,E2 -658.628} C_VEL
LIN {X 0,Y 601.38,Z 231.069,A -85,B 0,C 180,E1 -660.944,E2 -660.944} C_VEL
LIN {X 0,Y 601.384,Z 231.069,A -85,B 0,C 180,E1 -663.316,E2 -663.316} C_VEL
LIN {X 0,Y 601.393,Z 231.072,A -85,B 0,C 180,E1 -666.271,E2 -666.271} C_VEL
LIN {X 0,Y 601.385,Z 231.069,A -85,B 0,C 180,E1 -669.128,E2 -669.128} C_VEL
LIN {X 0,Y 601.387,Z 231.078,A -85,B 0,C 180,E1 -671.767,E2 -671.767} C_VEL
LIN {X 0,Y 601.372,Z 231.07,A -85,B 0,C 180,E1 -674.539,E2 -674.539} C_VEL
LIN {X 0,Y 601.412,Z 231.072,A -85,B 0,C 180,E1 -677.408,E2 -677.408} C_VEL
LIN {X 0,Y 601.366,Z 231.07,A -85,B 0,C 180,E1 -680.472,E2 -680.472} C_VEL
LIN {X 0,Y 601.391,Z 231.068,A -85,B 0,C 180,E1 -682.622,E2 -682.622} C_VEL
LIN {X 0,Y 601.412,Z 231.07,A -85,B 0,C 180,E1 -685.075,E2 -685.075} C_VEL
LIN {X 0,Y 601.411,Z 231.072,A -85,B 0,C 180,E1 -687.49,E2 -687.49} C_VEL
LIN {X 0,Y 601.389,Z 231.069,A -85,B 0,C 180,E1 -689.856,E2 -689.856} C_VEL
LIN {X 0,Y 601.366,Z 231.07,A -85,B 0,C 180,E1 -692.136,E2 -692.136} C_VEL
LIN {X 0,Y 601.385,Z 231.069,A -85,B 0,C 180,E1 -694.386,E2 -694.386} C_VEL
LIN {X 0,Y 601.384,Z 231.072,A -85,B 0,C 180,E1 -696.594,E2 -696.594} C_VEL
LIN {X 0,Y 601.396,Z 231.069,A -85,B 0,C 180,E1 -699.482,E2 -699.482} C_VEL
LIN {X 0,Y 601.366,Z 231.073,A -85,B 0,C 180,E1 -702.316,E2 -702.316} C_VEL
LIN {X 0,Y 601.391,Z 231.072,A -85,B 0,C 180,E1 -704.413,E2 -704.413} C_VEL
LIN {X 0,Y 601.391,Z 231.07,A -85,B 0,C 180,E1 -707.176,E2 -707.176} C_VEL
LIN {X 0,Y 601.391,Z 231.069,A -85,B 0,C 180,E1 -709.228,E2 -709.228} C_VEL
LIN {X 0,Y 601.383,Z 231.07,A -85,B 0,C 180,E1 -711.943,E2 -711.943} C_VEL
LIN {X 0,Y 601.419,Z 231.071,A -85,B 0,C 180,E1 -714.64,E2 -714.64} C_VEL
LIN {X 0,Y 601.396,Z 231.067,A -85,B 0,C 180,E1 -717.325,E2 -717.325} C_VEL
LIN {X 0,Y 601.421,Z 231.069,A -85,B 0,C 180,E1 -720.004,E2 -720.004} C_VEL
LIN {X 0,Y 601.425,Z 231.066,A -85,B 0,C 180,E1 -722.683,E2 -722.683} C_VEL
LIN {X 0,Y 601.383,Z 231.069,A -85,B 0,C 180,E1 -725.368,E2 -725.368} C_VEL
LIN {X 0,Y 601.427,Z 231.073,A -85,B 0,C 180,E1 -728.064,E2 -728.064} C_VEL
LIN {X 0,Y 601.383,Z 231.068,A -85,B 0,C 180,E1 -730.997,E2 -730.997} C_VEL
LIN {X 0,Y 601.392,Z 231.071,A -85,B 0,C 180,E1 -733.52,E2 -733.52} C_VEL
LIN {X 0,Y 601.408,Z 231.068,A -85,B 0,C 180,E1 -736.291,E2 -736.291} C_VEL
LIN {X 0,Y 601.399,Z 231.068,A -85,B 0,C 180,E1 -739.102,E2 -739.102} C_VEL
LIN {X 0,Y 601.389,Z 231.073,A -85,B 0,C 180,E1 -741.963,E2 -741.963} C_VEL
LIN {X 0,Y 601.379,Z 231.07,A -85,B 0,C 180,E1 -744.882,E2 -744.882} C_VEL
LIN {X 0,Y 601.398,Z 231.074,A -85,B 0,C 180,E1 -747.361,E2 -747.361} C_VEL
LIN {X 0,Y 601.401,Z 231.067,A -85,B 0,C 180,E1 -750.168,E2 -750.168} C_VEL
LIN {X 0,Y 601.391,Z 231.069,A -85,B 0,C 180,E1 -752.712,E2 -752.712} C_VEL
LIN {X 0,Y 601.377,Z 231.077,A -85,B 0,C 180,E1 -755.111,E2 -755.111} C_VEL
LIN {X 0,Y 601.433,Z 231.069,A -85,B 0,C 180,E1 -757.421,E2 -757.421} C_VEL
LIN {X 0,Y 601.38,Z 231.069,A -85,B 0,C 180,E1 -760,E2 -760} C_VEL
LIN {X 0,Y 601.376,Z 231.074,A -85,B 0,C 180,E1 -762.675,E2 -762.675} C_VEL
LIN {X 0,Y 601.403,Z 231.07,A -85,B 0,C 180,E1 -765.481,E2 -765.481} C_VEL
LIN {X 0,Y 601.407,Z 231.182,A -85,B 0,C 180,E1 -768.234,E2 -768.234} C_VEL
LIN {X 0,Y 601.452,Z 234.38,A -85,B 0,C 180,E1 -770.009,E2 -770.009} C_VEL
LIN {X 0,Y 601.443,Z 239.847,A -85,B 0,C 180,E1 -772.619,E2 -772.619} C_VEL
LIN {X 0,Y 601.444,Z 245.159,A -85,B 0,C 180,E1 -775.071,E2 -775.071} C_VEL
LIN {X 0,Y 601.413,Z 250.548,A -85,B 0,C 180,E1 -777.484,E2 -777.484} C_VEL
LIN {X 0,Y 601.434,Z 255.974,A -85,B 0,C 180,E1 -779.852,E2 -779.852} C_VEL
LIN {X 0,Y 601.404,Z 262.537,A -85,B 0,C 180,E1 -782.641,E2 -782.641} C_VEL
LIN {X 0,Y 601.398,Z 268.513,A -85,B 0,C 180,E1 -785.122,E2 -785.122} C_VEL
LIN {X 0,Y 601.378,Z 274.123,A -85,B 0,C 180,E1 -787.405,E2 -787.405} C_VEL
LIN {X 0,Y 601.372,Z 281.089,A -85,B 0,C 180,E1 -790.19,E2 -790.19} C_VEL
LIN {X 0,Y 601.342,Z 288.275,A -85,B 0,C 180,E1 -793.012,E2 -793.012} C_VEL
LIN {X 0,Y 601.352,Z 295.835,A -85,B 0,C 180,E1 -795.937,E2 -795.937} C_VEL
LIN {X 0,Y 601.368,Z 301.624,A -85,B 0,C 180,E1 -798.113,E2 -798.113} C_VEL
LIN {X 0,Y 601.591,Z 312.182,A -85,B 0,C 180,E1 -798.332,E2 -798.332} C_VEL
LIN {X 0,Y 601.53,Z 324.409,A -85,B 0,C 180,E1 -798.694,E2 -798.694} C_VEL
LIN {X 0,Y 601.454,Z 337.179,A -85,B 0,C 180,E1 -799.225,E2 -799.225} C_VEL
LIN {X 0,Y 601.46,Z 348.17,A -85,B 0,C 180,E1 -799.821,E2 -799.821} C_VEL
LIN {X 0,Y 601.455,Z 359.396,A -85,B 0,C 180,E1 -800.585,E2 -800.585} C_VEL
LIN {X 0,Y 601.423,Z 369.34,A -85,B 0,C 180,E1 -801.432,E2 -801.432} C_VEL
LIN {X 0,Y 601.418,Z 378.959,A -85,B 0,C 180,E1 -802.446,E2 -802.446} C_VEL
LIN {X 0,Y 601.371,Z 386.226,A -85,B 0,C 180,E1 -803.399,E2 -803.399} C_VEL
LIN {X 0,Y 601.372,Z 391.863,A -85,B 0,C 180,E1 -804.299,E2 -804.299} C_VEL
LIN {X 0,Y 601.336,Z 396.951,A -85,B 0,C 180,E1 -805.307,E2 -805.307} C_VEL
LIN {X 0,Y 601.368,Z 400.896,A -85,B 0,C 180,E1 -806.315,E2 -806.315} C_VEL
LIN {X 0,Y 601.325,Z 403.807,A -85,B 0,C 180,E1 -807.32,E2 -807.32} C_VEL
LIN {X 0,Y 601.343,Z 405.2,A -85,B 0,C 180,E1 -807.991,E2 -807.991} C_VEL
LIN {X 0,Y 601.339,Z 406.783,A -85,B 0,C 180,E1 -809.33,E2 -809.33} C_VEL
LIN {X 0,Y 601.335,Z 406.995,A -85,B 0,C 180,E1 -810,E2 -810} C_VEL
LIN {X 0,Y 601.348,Z 406.185,A -85,B 0,C 180,E1 -811.339,E2 -811.339} C_VEL
LIN {X 0,Y 601.343,Z 405.2,A -85,B 0,C 180,E1 -812.009,E2 -812.009} C_VEL
LIN {X 0,Y 601.325,Z 403.807,A -85,B 0,C 180,E1 -812.68,E2 -812.68} C_VEL
LIN {X 0,Y 601.368,Z 400.896,A -85,B 0,C 180,E1 -813.685,E2 -813.685} C_VEL
LIN {X 0,Y 601.336,Z 396.951,A -85,B 0,C 180,E1 -814.693,E2 -814.693} C_VEL
LIN {X 0,Y 601.372,Z 391.863,A -85,B 0,C 180,E1 -815.701,E2 -815.701} C_VEL
LIN {X 0,Y 601.383,Z 385.472,A -85,B 0,C 180,E1 -816.711,E2 -816.711} C_VEL
LIN {X 0,Y 601.396,Z 377.481,A -85,B 0,C 180,E1 -817.723,E2 -817.723} C_VEL
LIN {X 0,Y 601.423,Z 369.34,A -85,B 0,C 180,E1 -818.568,E2 -818.568} C_VEL
LIN {X 0,Y 601.455,Z 359.396,A -85,B 0,C 180,E1 -819.415,E2 -819.415} C_VEL
LIN {X 0,Y 601.46,Z 348.17,A -85,B 0,C 180,E1 -820.179,E2 -820.179} C_VEL
LIN {X 0,Y 601.454,Z 337.179,A -85,B 0,C 180,E1 -820.775,E2 -820.775} C_VEL
LIN {X 0,Y 601.532,Z 324.774,A -85,B 0,C 180,E1 -821.293,E2 -821.293} C_VEL
LIN {X 0,Y 601.591,Z 312.182,A -85,B 0,C 180,E1 -821.668,E2 -821.668} C_VEL
LIN {X 0,Y 601.368,Z 301.624,A -85,B 0,C 180,E1 -821.887,E2 -821.887} C_VEL
LIN {X 0,Y 601.338,Z 293.664,A -85,B 0,C 180,E1 -824.899,E2 -824.899} C_VEL
LIN {X 0,Y 601.356,Z 286.478,A -85,B 0,C 180,E1 -827.689,E2 -827.689} C_VEL
LIN {X 0,Y 601.366,Z 279.292,A -85,B 0,C 180,E1 -830.524,E2 -830.524} C_VEL
LIN {X 0,Y 601.388,Z 272.106,A -85,B 0,C 180,E1 -833.411,E2 -833.411} C_VEL
LIN {X 0,Y 601.397,Z 266.128,A -85,B 0,C 180,E1 -835.862,E2 -835.862} C_VEL
LIN {X 0,Y 601.423,Z 259.159,A -85,B 0,C 180,E1 -838.785,E2 -838.785} C_VEL
LIN {X 0,Y 601.444,Z 252.955,A -85,B 0,C 180,E1 -841.457,E2 -841.457} C_VEL
LIN {X 0,Y 601.425,Z 246.955,A -85,B 0,C 180,E1 -844.118,E2 -844.118} C_VEL
LIN {X 0,Y 601.439,Z 241.566,A -85,B 0,C 180,E1 -846.58,E2 -846.58} C_VEL
LIN {X 0,Y 601.445,Z 235.322,A -85,B 0,C 180,E1 -849.534,E2 -849.534} C_VEL
LIN {X 0,Y 601.451,Z 231.463,A -85,B 0,C 180,E1 -851.594,E2 -851.594} C_VEL
LIN {X 0,Y 601.407,Z 231.183,A -85,B 0,C 180,E1 -851.766,E2 -851.766} C_VEL
LIN {X 0,Y 601.402,Z 231.07,A -85,B 0,C 180,E1 -854.531,E2 -854.531} C_VEL
LIN {X 0,Y 601.376,Z 231.074,A -85,B 0,C 180,E1 -857.325,E2 -857.325} C_VEL
LIN {X 0,Y 601.38,Z 231.069,A -85,B 0,C 180,E1 -860,E2 -860} C_VEL
LIN {X 0,Y 601.436,Z 231.069,A -85,B 0,C 180,E1 -862.617,E2 -862.617} C_VEL
LIN {X 0,Y 601.384,Z 231.073,A -85,B 0,C 180,E1 -865.064,E2 -865.064} C_VEL
LIN {X 0,Y 601.389,Z 231.068,A -85,B 0,C 180,E1 -867.479,E2 -867.479} C_VEL
LIN {X 0,Y 601.402,Z 231.067,A -85,B 0,C 180,E1 -869.854,E2 -869.854} C_VEL
LIN {X 0,Y 601.407,Z 231.069,A -85,B 0,C 180,E1 -872.884,E2 -872.884} C_VEL
LIN {X 0,Y 601.379,Z 231.07,A -85,B 0,C 180,E1 -875.118,E2 -875.118} C_VEL
LIN {X 0,Y 601.389,Z 231.073,A -85,B 0,C 180,E1 -878.037,E2 -878.037} C_VEL
LIN {X 0,Y 601.399,Z 231.068,A -85,B 0,C 180,E1 -880.898,E2 -880.898} C_VEL
LIN {X 0,Y 601.408,Z 231.068,A -85,B 0,C 180,E1 -883.709,E2 -883.709} C_VEL
LIN {X 0,Y 601.392,Z 231.071,A -85,B 0,C 180,E1 -886.48,E2 -886.48} C_VEL
LIN {X 0,Y 601.371,Z 231.07,A -85,B 0,C 180,E1 -889.22,E2 -889.22} C_VEL
LIN {X 0,Y 601.427,Z 231.073,A -85,B 0,C 180,E1 -891.936,E2 -891.936} C_VEL
LIN {X 0,Y 601.383,Z 231.069,A -85,B 0,C 180,E1 -894.632,E2 -894.632} C_VEL
LIN {X 0,Y 601.425,Z 231.066,A -85,B 0,C 180,E1 -897.317,E2 -897.317} C_VEL
LIN {X 0,Y 601.421,Z 231.069,A -85,B 0,C 180,E1 -899.996,E2 -899.996} C_VEL
LIN {X 0,Y 601.396,Z 231.067,A -85,B 0,C 180,E1 -902.675,E2 -902.675} C_VEL
LIN {X 0,Y 601.419,Z 231.071,A -85,B 0,C 180,E1 -905.36,E2 -905.36} C_VEL
LIN {X 0,Y 601.383,Z 231.07,A -85,B 0,C 180,E1 -908.057,E2 -908.057} C_VEL
LIN {X 0,Y 601.443,Z 231.066,A -85,B 0,C 180,E1 -911.026,E2 -911.026} C_VEL
LIN {X 0,Y 601.373,Z 231.07,A -85,B 0,C 180,E1 -912.336,E2 -912.336} C_VEL
LIN {X 0,Y 600.711,Z 231.157,A -85,B 0,C 180,E1 -912.895,E2 -912.895} C_VEL
LIN {X 0,Y 597.861,Z 231.514,A -85,B 0,C 180,E1 -913.803,E2 -913.803} C_VEL
LIN {X 0,Y 595.45,Z 231.816,A -85,B 0,C 180,E1 -914.533,E2 -914.533} C_VEL
LIN {X 0,Y 594.413,Z 231.945,A -85,B 0,C 180,E1 -915.096,E2 -915.096} C_VEL
LIN {X 0,Y 594.327,Z 231.952,A -85,B 0,C 180,E1 -915.287,E2 -915.287} C_VEL
LIN {X 0,Y 594.316,Z 231.949,A -85,B 0,C 180,E1 -917.901,E2 -917.901} C_VEL
LIN {X 0,Y 594.376,Z 231.947,A -85,B 0,C 180,E1 -920.771,E2 -920.771} C_VEL
LIN {X 0,Y 594.348,Z 231.945,A -85,B 0,C 180,E1 -923.7,E2 -923.7} C_VEL
LIN {X 0,Y 594.355,Z 231.951,A -85,B 0,C 180,E1 -926.695,E2 -926.695} C_VEL
LIN {X 0,Y 594.35,Z 231.952,A -85,B 0,C 180,E1 -928.994,E2 -928.994} C_VEL
LIN {X 0,Y 594.338,Z 231.946,A -85,B 0,C 180,E1 -931.638,E2 -931.638} C_VEL
LIN {X 0,Y 594.362,Z 231.952,A -85,B 0,C 180,E1 -934.574,E2 -934.574} C_VEL
LIN {X 0,Y 594.344,Z 231.948,A -85,B 0,C 180,E1 -937.082,E2 -937.082} C_VEL
LIN {X 0,Y 594.318,Z 231.949,A -85,B 0,C 180,E1 -939.769,E2 -939.769} C_VEL
LIN {X 0,Y 594.355,Z 231.953,A -85,B 0,C 180,E1 -942.368,E2 -942.368} C_VEL
LIN {X 0,Y 594.311,Z 231.949,A -85,B 0,C 180,E1 -945.187,E2 -945.187} C_VEL
LIN {X 0,Y 594.343,Z 231.954,A -85,B 0,C 180,E1 -948.146,E2 -948.146} C_VEL
LIN {X 0,Y 594.336,Z 231.946,A -85,B 0,C 180,E1 -951.192,E2 -951.192} C_VEL
LIN {X 0,Y 594.346,Z 231.95,A -85,B 0,C 180,E1 -953.756,E2 -953.756} C_VEL
LIN {X 0,Y 594.338,Z 231.952,A -85,B 0,C 180,E1 -956.237,E2 -956.237} C_VEL
LIN {X 0,Y 594.334,Z 231.947,A -85,B 0,C 180,E1 -958.648,E2 -958.648} C_VEL
LIN {X 0,Y 594.336,Z 231.947,A -85,B 0,C 180,E1 -961.036,E2 -961.036} C_VEL
LIN {X 0,Y 594.339,Z 231.953,A -85,B 0,C 180,E1 -963.971,E2 -963.971} C_VEL
LIN {X 0,Y 594.346,Z 231.947,A -85,B 0,C 180,E1 -966.295,E2 -966.295} C_VEL
LIN {X 0,Y 594.365,Z 231.946,A -85,B 0,C 180,E1 -969.223,E2 -969.223} C_VEL
LIN {X 0,Y 594.327,Z 231.95,A -85,B 0,C 180,E1 -972.095,E2 -972.095} C_VEL
LIN {X 0,Y 594.318,Z 231.949,A -85,B 0,C 180,E1 -974.218,E2 -974.218} C_VEL
LIN {X 0,Y 594.35,Z 231.949,A -85,B 0,C 180,E1 -977.017,E2 -977.017} C_VEL
LIN {X 0,Y 594.343,Z 231.949,A -85,B 0,C 180,E1 -979.783,E2 -979.783} C_VEL
LIN {X 0,Y 594.353,Z 231.945,A -85,B 0,C 180,E1 -982.526,E2 -982.526} C_VEL
LIN {X 0,Y 594.356,Z 231.953,A -85,B 0,C 180,E1 -985.252,E2 -985.252} C_VEL
LIN {X 0,Y 594.326,Z 231.948,A -85,B 0,C 180,E1 -987.967,E2 -987.967} C_VEL
LIN {X 0,Y 594.378,Z 231.947,A -85,B 0,C 180,E1 -990.677,E2 -990.677} C_VEL
LIN {X 0,Y 594.336,Z 231.949,A -85,B 0,C 180,E1 -993.39,E2 -993.39} C_VEL
LIN {X 0,Y 594.341,Z 231.948,A -85,B 0,C 180,E1 -995.428,E2 -995.428} C_VEL
LIN {X 0,Y 594.353,Z 231.945,A -85,B 0,C 180,E1 -997.474,E2 -997.474} C_VEL
LIN {X 0,Y 594.343,Z 231.949,A -85,B 0,C 180,E1 -1000.217,E2 -1000.217} C_VEL
LIN {X 0,Y 594.35,Z 231.949,A -85,B 0,C 180,E1 -1002.983,E2 -1002.983} C_VEL
LIN {X 0,Y 594.318,Z 231.949,A -85,B 0,C 180,E1 -1005.782,E2 -1005.782} C_VEL
LIN {X 0,Y 594.351,Z 231.952,A -85,B 0,C 180,E1 -1008.618,E2 -1008.618} C_VEL
LIN {X 0,Y 594.319,Z 231.949,A -85,B 0,C 180,E1 -1011.505,E2 -1011.505} C_VEL
LIN {X 0,Y 594.346,Z 231.947,A -85,B 0,C 180,E1 -1013.705,E2 -1013.705} C_VEL
LIN {X 0,Y 594.331,Z 231.949,A -85,B 0,C 180,E1 -1016.702,E2 -1016.702} C_VEL
LIN {X 0,Y 594.334,Z 231.947,A -85,B 0,C 180,E1 -1019,E2 -1019} C_VEL
LIN {X 0,Y 594.34,Z 231.949,A -85,B 0,C 180,E1 -1021.65,E2 -1021.65} C_VEL
LIN {X 0,Y 594.34,Z 231.947,A -85,B 0,C 180,E1 -1024.582,E2 -1024.582} C_VEL
LIN {X 0,Y 594.329,Z 231.947,A -85,B 0,C 180,E1 -1027.09,E2 -1027.09} C_VEL
LIN {X 0,Y 594.336,Z 231.956,A -85,B 0,C 180,E1 -1029.78,E2 -1029.78} C_VEL
LIN {X 0,Y 594.319,Z 231.95,A -85,B 0,C 180,E1 -1032.379,E2 -1032.379} C_VEL
LIN {X 0,Y 594.312,Z 231.952,A -85,B 0,C 180,E1 -1035.195,E2 -1035.195} C_VEL
LIN {X 0,Y 594.355,Z 231.953,A -85,B 0,C 180,E1 -1037.632,E2 -1037.632} C_VEL
LIN {X 0,Y 594.331,Z 231.947,A -85,B 0,C 180,E1 -1040.324,E2 -1040.324} C_VEL
LIN {X 0,Y 594.344,Z 231.948,A -85,B 0,C 180,E1 -1042.918,E2 -1042.918} C_VEL
LIN {X 0,Y 594.343,Z 231.948,A -85,B 0,C 180,E1 -1045.865,E2 -1045.865} C_VEL
LIN {X 0,Y 594.332,Z 231.948,A -85,B 0,C 180,E1 -1048.654,E2 -1048.654} C_VEL
LIN {X 0,Y 594.355,Z 231.952,A -85,B 0,C 180,E1 -1051.045,E2 -1051.045} C_VEL
LIN {X 0,Y 594.341,Z 231.946,A -85,B 0,C 180,E1 -1053.984,E2 -1053.984} C_VEL
LIN {X 0,Y 594.348,Z 231.945,A -85,B 0,C 180,E1 -1056.3,E2 -1056.3} C_VEL
LIN {X 0,Y 594.376,Z 231.947,A -85,B 0,C 180,E1 -1059.229,E2 -1059.229} C_VEL
LIN {X 0,Y 594.316,Z 231.949,A -85,B 0,C 180,E1 -1062.099,E2 -1062.099} C_VEL
LIN {X 0,Y 594.337,Z 231.948,A -85,B 0,C 180,E1 -1064.223,E2 -1064.223} C_VEL
LIN {X 0,Y 594.34,Z 231.951,A -85,B 0,C 180,E1 -1067.021,E2 -1067.021} C_VEL
LIN {X 0,Y 594.37,Z 231.945,A -85,B 0,C 180,E1 -1069.099,E2 -1069.099} C_VEL
LIN {X 0,Y 594.336,Z 231.947,A -85,B 0,C 180,E1 -1071.847,E2 -1071.847} C_VEL
LIN {X 0,Y 594.38,Z 231.949,A -85,B 0,C 180,E1 -1074.576,E2 -1074.576} C_VEL
LIN {X 0,Y 594.366,Z 231.943,A -85,B 0,C 180,E1 -1077.293,E2 -1077.293} C_VEL
LIN {X 0,Y 594.391,Z 231.944,A -85,B 0,C 180,E1 -1080.004,E2 -1080.004} C_VEL
LIN {X 0,Y 594.388,Z 231.943,A -85,B 0,C 180,E1 -1082.715,E2 -1082.715} C_VEL
LIN {X 0,Y 594.351,Z 231.945,A -85,B 0,C 180,E1 -1085.432,E2 -1085.432} C_VEL
LIN {X 0,Y 594.371,Z 231.951,A -85,B 0,C 180,E1 -1088.161,E2 -1088.161} C_VEL
LIN {X 0,Y 594.36,Z 231.943,A -85,B 0,C 180,E1 -1091.064,E2 -1091.064} C_VEL
LIN {X 0,Y 594.364,Z 231.949,A -85,B 0,C 180,E1 -1093.683,E2 -1093.683} C_VEL
LIN {X 0,Y 594.33,Z 231.947,A -85,B 0,C 180,E1 -1096.702,E2 -1096.702} C_VEL
LIN {X 0,Y 594.353,Z 231.948,A -85,B 0,C 180,E1 -1099.338,E2 -1099.338} C_VEL
LIN {X 0,Y 594.347,Z 231.952,A -85,B 0,C 180,E1 -1101.507,E2 -1101.507} C_VEL
LIN {X 0,Y 594.345,Z 231.945,A -85,B 0,C 180,E1 -1104.451,E2 -1104.451} C_VEL
LIN {X 0,Y 594.355,Z 231.944,A -85,B 0,C 180,E1 -1106.704,E2 -1106.704} C_VEL
LIN {X 0,Y 594.355,Z 231.948,A -85,B 0,C 180,E1 -1109.78,E2 -1109.78} C_VEL
LIN {X 0,Y 594.341,Z 231.946,A -85,B 0,C 180,E1 -1112.151,E2 -1112.151} C_VEL
LIN {X 0,Y 594.36,Z 231.944,A -85,B 0,C 180,E1 -1114.584,E2 -1114.584} C_VEL
LIN {X 0,Y 594.38,Z 231.945,A -85,B 0,C 180,E1 -1117.609,E2 -1117.609} C_VEL
LIN {X 0,Y 594.344,Z 231.948,A -85,B 0,C 180,E1 -1120.571,E2 -1120.571} C_VEL
LIN {X 0,Y 594.347,Z 231.952,A -85,B 0,C 180,E1 -1123.303,E2 -1123.303} C_VEL
LIN {X 0,Y 594.346,Z 231.948,A -85,B 0,C 180,E1 -1126.165,E2 -1126.165} C_VEL
LIN {X 0,Y 594.343,Z 231.953,A -85,B 0,C 180,E1 -1127.623,E2 -1127.623} C_VEL
LIN {X 0,Y 594.492,Z 233.037,A -85,B 0,C 180,E1 -1128.547,E2 -1128.547} C_VEL
LIN {X 0,Y 594.443,Z 238.159,A -85,B 0,C 180,E1 -1131.291,E2 -1131.291} C_VEL
LIN {X 0,Y 594.406,Z 243.362,A -85,B 0,C 180,E1 -1133.76,E2 -1133.76} C_VEL
LIN {X 0,Y 594.396,Z 248.752,A -85,B 0,C 180,E1 -1136.241,E2 -1136.241} C_VEL
LIN {X 0,Y 594.397,Z 254.141,A -85,B 0,C 180,E1 -1138.652,E2 -1138.652} C_VEL
LIN {X 0,Y 594.382,Z 259.628,A -85,B 0,C 180,E1 -1141.044,E2 -1141.044} C_VEL
LIN {X 0,Y 594.343,Z 266.717,A -85,B 0,C 180,E1 -1144.055,E2 -1144.055} C_VEL
LIN {X 0,Y 594.312,Z 272.106,A -85,B 0,C 180,E1 -1146.293,E2 -1146.293} C_VEL
LIN {X 0,Y 594.332,Z 279.292,A -85,B 0,C 180,E1 -1149.222,E2 -1149.222} C_VEL
LIN {X 0,Y 594.269,Z 286.478,A -85,B 0,C 180,E1 -1152.093,E2 -1152.093} C_VEL
LIN {X 0,Y 594.265,Z 293.664,A -85,B 0,C 180,E1 -1154.92,E2 -1154.92} C_VEL
LIN {X 0,Y 594.272,Z 301.468,A -85,B 0,C 180,E1 -1157.948,E2 -1157.948} C_VEL
LIN {X 0,Y 594.653,Z 306.395,A -85,B 0,C 180,E1 -1158.064,E2 -1158.064} C_VEL
LIN {X 0,Y 594.62,Z 318.513,A -85,B 0,C 180,E1 -1158.366,E2 -1158.366} C_VEL
LIN {X 0,Y 594.527,Z 330.726,A -85,B 0,C 180,E1 -1158.805,E2 -1158.805} C_VEL
LIN {X 0,Y 594.471,Z 342.208,A -85,B 0,C 180,E1 -1159.355,E2 -1159.355} C_VEL
LIN {X 0,Y 594.458,Z 353.479,A -85,B 0,C 180,E1 -1160.043,E2 -1160.043} C_VEL
LIN {X 0,Y 594.406,Z 363.647,A -85,B 0,C 180,E1 -1160.815,E2 -1160.815} C_VEL
LIN {X 0,Y 594.373,Z 372.78,A -85,B 0,C 180,E1 -1161.672,E2 -1161.672} C_VEL
LIN {X 0,Y 594.317,Z 381.684,A -85,B 0,C 180,E1 -1162.697,E2 -1162.697} C_VEL
LIN {X 0,Y 594.281,Z 388.178,A -85,B 0,C 180,E1 -1163.617,E2 -1163.617} C_VEL
LIN {X 0,Y 594.289,Z 393.681,A -85,B 0,C 180,E1 -1164.571,E2 -1164.571} C_VEL
LIN {X 0,Y 594.27,Z 398.373,A -85,B 0,C 180,E1 -1165.591,E2 -1165.591} C_VEL
LIN {X 0,Y 594.267,Z 401.959,A -85,B 0,C 180,E1 -1166.61,E2 -1166.61} C_VEL
LIN {X 0,Y 594.226,Z 403.805,A -85,B 0,C 180,E1 -1167.288,E2 -1167.288} C_VEL
LIN {X 0,Y 594.242,Z 405.199,A -85,B 0,C 180,E1 -1167.967,E2 -1167.967} C_VEL
LIN {X 0,Y 594.239,Z 406.783,A -85,B 0,C 180,E1 -1169.322,E2 -1169.322} C_VEL
LIN {X 0,Y 594.236,Z 406.991,A -85,B 0,C 180,E1 -1170,E2 -1170} C_VEL
LIN {X 0,Y 594.247,Z 406.186,A -85,B 0,C 180,E1 -1171.355,E2 -1171.355} C_VEL
LIN {X 0,Y 594.242,Z 405.199,A -85,B 0,C 180,E1 -1172.033,E2 -1172.033} C_VEL
LIN {X 0,Y 594.226,Z 403.805,A -85,B 0,C 180,E1 -1172.712,E2 -1172.712} C_VEL
LIN {X 0,Y 594.289,Z 400.894,A -85,B 0,C 180,E1 -1173.729,E2 -1173.729} C_VEL
LIN {X 0,Y 594.241,Z 396.949,A -85,B 0,C 180,E1 -1174.749,E2 -1174.749} C_VEL
LIN {X 0,Y 594.299,Z 391.858,A -85,B 0,C 180,E1 -1175.769,E2 -1175.769} C_VEL
LIN {X 0,Y 594.317,Z 385.471,A -85,B 0,C 180,E1 -1176.791,E2 -1176.791} C_VEL
LIN {X 0,Y 594.347,Z 377.482,A -85,B 0,C 180,E1 -1177.815,E2 -1177.815} C_VEL
LIN {X 0,Y 594.378,Z 369.342,A -85,B 0,C 180,E1 -1178.671,E2 -1178.671} C_VEL
LIN {X 0,Y 594.419,Z 359.39,A -85,B 0,C 180,E1 -1179.528,E2 -1179.528} C_VEL
LIN {X 0,Y 594.447,Z 348.171,A -85,B 0,C 180,E1 -1180.301,E2 -1180.301} C_VEL
LIN {X 0,Y 594.507,Z 336.06,A -85,B 0,C 180,E1 -1180.958,E2 -1180.958} C_VEL
LIN {X 0,Y 594.55,Z 323.79,A -85,B 0,C 180,E1 -1181.461,E2 -1181.461} C_VEL
LIN {X 0,Y 594.662,Z 311.264,A -85,B 0,C 180,E1 -1181.828,E2 -1181.828} C_VEL
LIN {X 0,Y 594.396,Z 302.604,A -85,B 0,C 180,E1 -1182.012,E2 -1182.012} C_VEL
LIN {X 0,Y 594.272,Z 301.468,A -85,B 0,C 180,E1 -1182.052,E2 -1182.052} C_VEL
LIN {X 0,Y 594.265,Z 293.664,A -85,B 0,C 180,E1 -1185.08,E2 -1185.08} C_VEL
LIN {X 0,Y 594.268,Z 286.478,A -85,B 0,C 180,E1 -1187.907,E2 -1187.907} C_VEL
LIN {X 0,Y 594.332,Z 279.292,A -85,B 0,C 180,E1 -1190.778,E2 -1190.778} C_VEL
LIN {X 0,Y 594.312,Z 272.106,A -85,B 0,C 180,E1 -1193.707,E2 -1193.707} C_VEL
LIN {X 0,Y 594.336,Z 266.56,A -85,B 0,C 180,E1 -1196.011,E2 -1196.011} C_VEL
LIN {X 0,Y 594.38,Z 259.531,A -85,B 0,C 180,E1 -1198.998,E2 -1198.998} C_VEL
LIN {X 0,Y 594.394,Z 253.474,A -85,B 0,C 180,E1 -1201.643,E2 -1201.643} C_VEL
LIN {X 0,Y 594.398,Z 246.955,A -85,B 0,C 180,E1 -1204.578,E2 -1204.578} C_VEL
LIN {X 0,Y 594.419,Z 241.566,A -85,B 0,C 180,E1 -1207.083,E2 -1207.083} C_VEL
LIN {X 0,Y 594.466,Z 236.053,A -85,B 0,C 180,E1 -1209.783,E2 -1209.783} C_VEL
LIN {X 0,Y 594.492,Z 233.039,A -85,B 0,C 180,E1 -1211.453,E2 -1211.453} C_VEL
LIN {X 0,Y 594.343,Z 231.953,A -85,B 0,C 180,E1 -1212.377,E2 -1212.377} C_VEL
LIN {X 0,Y 594.342,Z 231.954,A -85,B 0,C 180,E1 -1215.192,E2 -1215.192} C_VEL
LIN {X 0,Y 594.364,Z 231.944,A -85,B 0,C 180,E1 -1218.153,E2 -1218.153} C_VEL
LIN {X 0,Y 594.359,Z 231.947,A -85,B 0,C 180,E1 -1221.297,E2 -1221.297} C_VEL
LIN {X 0,Y 594.341,Z 231.946,A -85,B 0,C 180,E1 -1223.752,E2 -1223.752} C_VEL
LIN {X 0,Y 594.361,Z 231.946,A -85,B 0,C 180,E1 -1226.235,E2 -1226.235} C_VEL
LIN {X 0,Y 594.362,Z 231.953,A -85,B 0,C 180,E1 -1228.647,E2 -1228.647} C_VEL
LIN {X 0,Y 594.371,Z 231.945,A -85,B 0,C 180,E1 -1231.043,E2 -1231.043} C_VEL
LIN {X 0,Y 594.368,Z 231.946,A -85,B 0,C 180,E1 -1234.053,E2 -1234.053} C_VEL
LIN {X 0,Y 594.347,Z 231.946,A -85,B 0,C 180,E1 -1237.029,E2 -1237.029} C_VEL
LIN {X 0,Y 594.353,Z 231.949,A -85,B 0,C 180,E1 -1239.943,E2 -1239.943} C_VEL
LIN {X 0,Y 594.324,Z 231.949,A -85,B 0,C 180,E1 -1242.802,E2 -1242.802} C_VEL
LIN {X 0,Y 594.384,Z 231.946,A -85,B 0,C 180,E1 -1245.824,E2 -1245.824} C_VEL
LIN {X 0,Y 594.368,Z 231.946,A -85,B 0,C 180,E1 -1248.4,E2 -1248.4} C_VEL
LIN {X 0,Y 594.356,Z 231.944,A -85,B 0,C 180,E1 -1251.154,E2 -1251.154} C_VEL
LIN {X 0,Y 594.344,Z 231.955,A -85,B 0,C 180,E1 -1253.887,E2 -1253.887} C_VEL
LIN {X 0,Y 594.34,Z 231.954,A -85,B 0,C 180,E1 -1255.928,E2 -1255.928} C_VEL
LIN {X 0,Y 594.375,Z 231.948,A -85,B 0,C 180,E1 -1257.963,E2 -1257.963} C_VEL
LIN {X 0,Y 594.391,Z 231.944,A -85,B 0,C 180,E1 -1259.996,E2 -1259.996} C_VEL
LIN {X 0,Y 594.366,Z 231.943,A -85,B 0,C 180,E1 -1262.707,E2 -1262.707} C_VEL
LIN {X 0,Y 594.38,Z 231.949,A -85,B 0,C 180,E1 -1265.424,E2 -1265.424} C_VEL
LIN {X 0,Y 594.336,Z 231.947,A -85,B 0,C 180,E1 -1268.153,E2 -1268.153} C_VEL
LIN {X 0,Y 594.416,Z 231.942,A -85,B 0,C 180,E1 -1271.091,E2 -1271.091} C_VEL
LIN {X 0,Y 594.32,Z 231.948,A -85,B 0,C 180,E1 -1274.151,E2 -1274.151} C_VEL
LIN {X 0,Y 594.327,Z 231.952,A -85,B 0,C 180,E1 -1275.287,E2 -1275.287} C_VEL
LIN {X 0,Y 593.654,Z 232.034,A -85,B 0,C 180,E1 -1275.853,E2 -1275.853} C_VEL
LIN {X 0,Y 590.785,Z 232.392,A -85,B 0,C 180,E1 -1276.771,E2 -1276.771} C_VEL
LIN {X 0,Y 588.372,Z 232.694,A -85,B 0,C 180,E1 -1277.509,E2 -1277.509} C_VEL
LIN {X 0,Y 587.349,Z 232.817,A -85,B 0,C 180,E1 -1278.079,E2 -1278.079} C_VEL
LIN {X 0,Y 587.273,Z 232.826,A -85,B 0,C 180,E1 -1278.272,E2 -1278.272} C_VEL
LIN {X 0,Y 587.303,Z 232.832,A -85,B 0,C 180,E1 -1281.033,E2 -1281.033} C_VEL
LIN {X 0,Y 587.288,Z 232.83,A -85,B 0,C 180,E1 -1283.254,E2 -1283.254} C_VEL
LIN {X 0,Y 587.295,Z 232.825,A -85,B 0,C 180,E1 -1285.512,E2 -1285.512} C_VEL
LIN {X 0,Y 587.314,Z 232.821,A -85,B 0,C 180,E1 -1287.813,E2 -1287.813} C_VEL
LIN {X 0,Y 587.3,Z 232.828,A -85,B 0,C 180,E1 -1290.505,E2 -1290.505} C_VEL
LIN {X 0,Y 587.29,Z 232.825,A -85,B 0,C 180,E1 -1293.392,E2 -1293.392} C_VEL
LIN {X 0,Y 587.316,Z 232.821,A -85,B 0,C 180,E1 -1295.891,E2 -1295.891} C_VEL
LIN {X 0,Y 587.288,Z 232.833,A -85,B 0,C 180,E1 -1298.475,E2 -1298.475} C_VEL
LIN {X 0,Y 587.29,Z 232.825,A -85,B 0,C 180,E1 -1301.152,E2 -1301.152} C_VEL
LIN {X 0,Y 587.284,Z 232.828,A -85,B 0,C 180,E1 -1303.945,E2 -1303.945} C_VEL
LIN {X 0,Y 587.272,Z 232.828,A -85,B 0,C 180,E1 -1306.877,E2 -1306.877} C_VEL
LIN {X 0,Y 587.278,Z 232.828,A -85,B 0,C 180,E1 -1309.744,E2 -1309.744} C_VEL
LIN {X 0,Y 587.294,Z 232.829,A -85,B 0,C 180,E1 -1312.389,E2 -1312.389} C_VEL
LIN {X 0,Y 587.293,Z 232.824,A -85,B 0,C 180,E1 -1314.943,E2 -1314.943} C_VEL
LIN {X 0,Y 587.289,Z 232.826,A -85,B 0,C 180,E1 -1317.419,E2 -1317.419} C_VEL
LIN {X 0,Y 587.315,Z 232.83,A -85,B 0,C 180,E1 -1319.829,E2 -1319.829} C_VEL
LIN {X 0,Y 587.289,Z 232.827,A -85,B 0,C 180,E1 -1322.304,E2 -1322.304} C_VEL
LIN {X 0,Y 587.306,Z 232.825,A -85,B 0,C 180,E1 -1325.24,E2 -1325.24} C_VEL
LIN {X 0,Y 587.316,Z 232.828,A -85,B 0,C 180,E1 -1327.486,E2 -1327.486} C_VEL
LIN {X 0,Y 587.291,Z 232.824,A -85,B 0,C 180,E1 -1330.424,E2 -1330.424} C_VEL
LIN {X 0,Y 587.323,Z 232.827,A -85,B 0,C 180,E1 -1333.311,E2 -1333.311} C_VEL
LIN {X 0,Y 587.301,Z 232.824,A -85,B 0,C 180,E1 -1336.153,E2 -1336.153} C_VEL
LIN {X 0,Y 587.3,Z 232.827,A -85,B 0,C 180,E1 -1338.962,E2 -1338.962} C_VEL
LIN {X 0,Y 587.315,Z 232.824,A -85,B 0,C 180,E1 -1341.744,E2 -1341.744} C_VEL
LIN {X 0,Y 587.27,Z 232.828,A -85,B 0,C 180,E1 -1343.817,E2 -1343.817} C_VEL
LIN {X 0,Y 587.253,Z 232.83,A -85,B 0,C 180,E1 -1345.882,E2 -1345.882} C_VEL
LIN {X 0,Y 587.297,Z 232.824,A -85,B 0,C 180,E1 -1347.943,E2 -1347.943} C_VEL
LIN {X 0,Y 587.346,Z 232.823,A -85,B 0,C 180,E1 -1350.686,E2 -1350.686} C_VEL
LIN {X 0,Y 587.286,Z 232.827,A -85,B 0,C 180,E1 -1353.43,E2 -1353.43} C_VEL
LIN {X 0,Y 587.304,Z 232.824,A -85,B 0,C 180,E1 -1355.493,E2 -1355.493} C_VEL
LIN {X 0,Y 587.317,Z 232.822,A -85,B 0,C 180,E1 -1357.564,E2 -1357.564} C_VEL
LIN {X 0,Y 587.294,Z 232.828,A -85,B 0,C 180,E1 -1360.341,E2 -1360.341} C_VEL
LIN {X 0,Y 587.29,Z 232.827,A -85,B 0,C 180,E1 -1363.142,E2 -1363.142} C_VEL
LIN {X 0,Y 587.282,Z 232.828,A -85,B 0,C 180,E1 -1365.976,E2 -1365.976} C_VEL
LIN {X 0,Y 587.312,Z 232.825,A -85,B 0,C 180,E1 -1368.85,E2 -1368.85} C_VEL
LIN {X 0,Y 587.28,Z 232.827,A -85,B 0,C 180,E1 -1371.775,E2 -1371.775} C_VEL
LIN {X 0,Y 587.315,Z 232.826,A -85,B 0,C 180,E1 -1374.589,E2 -1374.589} C_VEL
LIN {X 0,Y 587.278,Z 232.826,A -85,B 0,C 180,E1 -1377.048,E2 -1377.048} C_VEL
LIN {X 0,Y 587.306,Z 232.823,A -85,B 0,C 180,E1 -1379.381,E2 -1379.381} C_VEL
LIN {X 0,Y 587.304,Z 232.829,A -85,B 0,C 180,E1 -1381.842,E2 -1381.842} C_VEL
LIN {X 0,Y 587.305,Z 232.826,A -85,B 0,C 180,E1 -1384.354,E2 -1384.354} C_VEL
LIN {X 0,Y 587.296,Z 232.823,A -85,B 0,C 180,E1 -1386.75,E2 -1386.75} C_VEL
LIN {X 0,Y 587.3,Z 232.826,A -85,B 0,C 180,E1 -1389.362,E2 -1389.362} C_VEL
LIN {X 0,Y 587.281,Z 232.829,A -85,B 0,C 180,E1 -1392.112,E2 -1392.112} C_VEL
LIN {X 0,Y 587.264,Z 232.828,A -85,B 0,C 180,E1 -1394.915,E2 -1394.915} C_VEL
LIN {X 0,Y 587.305,Z 232.826,A -85,B 0,C 180,E1 -1397.932,E2 -1397.932} C_VEL
LIN {X 0,Y 587.281,Z 232.829,A -85,B 0,C 180,E1 -1401.063,E2 -1401.063} C_VEL
LIN {X 0,Y 587.312,Z 232.829,A -85,B 0,C 180,E1 -1403.296,E2 -1403.296} C_VEL
LIN {X 0,Y 587.308,Z 232.825,A -85,B 0,C 180,E1 -1405.784,E2 -1405.784} C_VEL
LIN {X 0,Y 587.305,Z 232.822,A -85,B 0,C 180,E1 -1408.236,E2 -1408.236} C_VEL
LIN {X 0,Y 587.318,Z 232.825,A -85,B 0,C 180,E1 -1410.87,E2 -1410.87} C_VEL
LIN {X 0,Y 587.303,Z 232.824,A -85,B 0,C 180,E1 -1413.726,E2 -1413.726} C_VEL
LIN {X 0,Y 587.29,Z 232.824,A -85,B 0,C 180,E1 -1415.997,E2 -1415.997} C_VEL
LIN {X 0,Y 587.288,Z 232.825,A -85,B 0,C 180,E1 -1418.23,E2 -1418.23} C_VEL
LIN {X 0,Y 587.32,Z 232.826,A -85,B 0,C 180,E1 -1421.156,E2 -1421.156} C_VEL
LIN {X 0,Y 587.292,Z 232.824,A -85,B 0,C 180,E1 -1424.029,E2 -1424.029} C_VEL
LIN {X 0,Y 587.29,Z 232.831,A -85,B 0,C 180,E1 -1426.863,E2 -1426.863} C_VEL
LIN {X 0,Y 587.354,Z 232.821,A -85,B 0,C 180,E1 -1428.967,E2 -1428.967} C_VEL
LIN {X 0,Y 587.302,Z 232.823,A -85,B 0,C 180,E1 -1431.748,E2 -1431.748} C_VEL
LIN {X 0,Y 587.342,Z 232.827,A -85,B 0,C 180,E1 -1434.511,E2 -1434.511} C_VEL
LIN {X 0,Y 587.336,Z 232.818,A -85,B 0,C 180,E1 -1437.261,E2 -1437.261} C_VEL
LIN {X 0,Y 587.36,Z 232.82,A -85,B 0,C 180,E1 -1440.004,E2 -1440.004} C_VEL
LIN {X 0,Y 587.352,Z 232.819,A -85,B 0,C 180,E1 -1442.747,E2 -1442.747} C_VEL
LIN {X 0,Y 587.32,Z 232.821,A -85,B 0,C 180,E1 -1445.497,E2 -1445.497} C_VEL
LIN {X 0,Y 587.331,Z 232.826,A -85,B 0,C 180,E1 -1448.259,E2 -1448.259} C_VEL
LIN {X 0,Y 587.327,Z 232.82,A -85,B 0,C 180,E1 -1451.128,E2 -1451.128} C_VEL
LIN {X 0,Y 587.347,Z 232.826,A -85,B 0,C 180,E1 -1453.849,E2 -1453.849} C_VEL
LIN {X 0,Y 587.283,Z 232.825,A -85,B 0,C 180,E1 -1456.796,E2 -1456.796} C_VEL
LIN {X 0,Y 587.298,Z 232.83,A -85,B 0,C 180,E1 -1459.58,E2 -1459.58} C_VEL
LIN {X 0,Y 587.305,Z 232.83,A -85,B 0,C 180,E1 -1461.778,E2 -1461.778} C_VEL
LIN {X 0,Y 587.303,Z 232.823,A -85,B 0,C 180,E1 -1464.763,E2 -1464.763} C_VEL
LIN {X 0,Y 587.298,Z 232.83,A -85,B 0,C 180,E1 -1467.685,E2 -1467.685} C_VEL
LIN {X 0,Y 587.313,Z 232.822,A -85,B 0,C 180,E1 -1470.174,E2 -1470.174} C_VEL
LIN {X 0,Y 587.325,Z 232.82,A -85,B 0,C 180,E1 -1472.582,E2 -1472.582} C_VEL
LIN {X 0,Y 587.303,Z 232.829,A -85,B 0,C 180,E1 -1475.06,E2 -1475.06} C_VEL
LIN {X 0,Y 587.319,Z 232.822,A -85,B 0,C 180,E1 -1477.837,E2 -1477.837} C_VEL
LIN {X 0,Y 587.296,Z 232.824,A -85,B 0,C 180,E1 -1480.258,E2 -1480.258} C_VEL
LIN {X 0,Y 587.293,Z 232.833,A -85,B 0,C 180,E1 -1483.117,E2 -1483.117} C_VEL
LIN {X 0,Y 587.302,Z 232.826,A -85,B 0,C 180,E1 -1486.049,E2 -1486.049} C_VEL
LIN {X 0,Y 587.292,Z 232.833,A -85,B 0,C 180,E1 -1486.993,E2 -1486.993} C_VEL
LIN {X 0,Y 587.396,Z 233.38,A -85,B 0,C 180,E1 -1487.932,E2 -1487.932} C_VEL
LIN {X 0,Y 587.491,Z 236.524,A -85,B 0,C 180,E1 -1489.761,E2 -1489.761} C_VEL
LIN {X 0,Y 587.4,Z 241.566,A -85,B 0,C 180,E1 -1492.397,E2 -1492.397} C_VEL
LIN {X 0,Y 587.374,Z 246.955,A -85,B 0,C 180,E1 -1494.948,E2 -1494.948} C_VEL
LIN {X 0,Y 587.345,Z 252.345,A -85,B 0,C 180,E1 -1497.422,E2 -1497.422} C_VEL
LIN {X 0,Y 587.337,Z 257.734,A -85,B 0,C 180,E1 -1499.831,E2 -1499.831} C_VEL
LIN {X 0,Y 587.302,Z 263.443,A -85,B 0,C 180,E1 -1502.318,E2 -1502.318} C_VEL
LIN {X 0,Y 587.296,Z 270.31,A -85,B 0,C 180,E1 -1505.239,E2 -1505.239} C_VEL
LIN {X 0,Y 587.25,Z 277.496,A -85,B 0,C 180,E1 -1508.223,E2 -1508.223} C_VEL
LIN {X 0,Y 587.243,Z 284.682,A -85,B 0,C 180,E1 -1511.148,E2 -1511.148} C_VEL
LIN {X 0,Y 587.187,Z 291.868,A -85,B 0,C 180,E1 -1514.021,E2 -1514.021} C_VEL
LIN {X 0,Y 587.159,Z 299.054,A -85,B 0,C 180,E1 -1516.855,E2 -1516.855} C_VEL
LIN {X 0,Y 587.151,Z 301.579,A -85,B 0,C 180,E1 -1517.821,E2 -1517.821} C_VEL
LIN {X 0,Y 587.723,Z 306.399,A -85,B 0,C 180,E1 -1517.921,E2 -1517.921} C_VEL
LIN {X 0,Y 587.687,Z 318.514,A -85,B 0,C 180,E1 -1518.227,E2 -1518.227} C_VEL
LIN {X 0,Y 587.563,Z 330.456,A -85,B 0,C 180,E1 -1518.66,E2 -1518.66} C_VEL
LIN {X 0,Y 587.497,Z 342.207,A -85,B 0,C 180,E1 -1519.227,E2 -1519.227} C_VEL
LIN {X 0,Y 587.456,Z 353.48,A -85,B 0,C 180,E1 -1519.924,E2 -1519.924} C_VEL
LIN {X 0,Y 587.385,Z 363.646,A -85,B 0,C 180,E1 -1520.705,E2 -1520.705} C_VEL
LIN {X 0,Y 587.331,Z 372.776,A -85,B 0,C 180,E1 -1521.571,E2 -1521.571} C_VEL
LIN {X 0,Y 587.26,Z 381.682,A -85,B 0,C 180,E1 -1522.609,E2 -1522.609} C_VEL
LIN {X 0,Y 587.195,Z 388.759,A -85,B 0,C 180,E1 -1523.629,E2 -1523.629} C_VEL
LIN {X 0,Y 587.211,Z 393.681,A -85,B 0,C 180,E1 -1524.506,E2 -1524.506} C_VEL
LIN {X 0,Y 587.189,Z 398.374,A -85,B 0,C 180,E1 -1525.538,E2 -1525.538} C_VEL
LIN {X 0,Y 587.194,Z 401.96,A -85,B 0,C 180,E1 -1526.569,E2 -1526.569} C_VEL
LIN {X 0,Y 587.132,Z 403.803,A -85,B 0,C 180,E1 -1527.256,E2 -1527.256} C_VEL
LIN {X 0,Y 587.141,Z 405.197,A -85,B 0,C 180,E1 -1527.942,E2 -1527.942} C_VEL
LIN {X 0,Y 587.147,Z 406.186,A -85,B 0,C 180,E1 -1528.628,E2 -1528.628} C_VEL
LIN {X 0,Y 587.137,Z 406.987,A -85,B 0,C 180,E1 -1530,E2 -1530} C_VEL
LIN {X 0,Y 587.147,Z 406.186,A -85,B 0,C 180,E1 -1531.372,E2 -1531.372} C_VEL
LIN {X 0,Y 587.141,Z 405.197,A -85,B 0,C 180,E1 -1532.058,E2 -1532.058} C_VEL
LIN {X 0,Y 587.132,Z 403.803,A -85,B 0,C 180,E1 -1532.744,E2 -1532.744} C_VEL
LIN {X 0,Y 587.213,Z 400.892,A -85,B 0,C 180,E1 -1533.774,E2 -1533.774} C_VEL
LIN {X 0,Y 587.147,Z 396.947,A -85,B 0,C 180,E1 -1534.806,E2 -1534.806} C_VEL
LIN {X 0,Y 587.229,Z 391.853,A -85,B 0,C 180,E1 -1535.839,E2 -1535.839} C_VEL
LIN {X 0,Y 587.232,Z 385.469,A -85,B 0,C 180,E1 -1536.874,E2 -1536.874} C_VEL
LIN {X 0,Y 587.288,Z 377.484,A -85,B 0,C 180,E1 -1537.91,E2 -1537.91} C_VEL
LIN {X 0,Y 587.336,Z 369.343,A -85,B 0,C 180,E1 -1538.775,E2 -1538.775} C_VEL
LIN {X 0,Y 587.39,Z 359.384,A -85,B 0,C 180,E1 -1539.643,E2 -1539.643} C_VEL
LIN {X 0,Y 587.44,Z 349.57,A -85,B 0,C 180,E1 -1540.338,E2 -1540.338} C_VEL
LIN {X 0,Y 587.494,Z 338.933,A -85,B 0,C 180,E1 -1540.947,E2 -1540.947} C_VEL
LIN {X 0,Y 587.573,Z 326.647,A -85,B 0,C 180,E1 -1541.493,E2 -1541.493} C_VEL
LIN {X 0,Y 587.713,Z 313.919,A -85,B 0,C 180,E1 -1541.904,E2 -1541.904} C_VEL
LIN {X 0,Y 587.563,Z 304.116,A -85,B 0,C 180,E1 -1542.126,E2 -1542.126} C_VEL
LIN {X 0,Y 587.146,Z 301.468,A -85,B 0,C 180,E1 -1542.201,E2 -1542.201} C_VEL
LIN {X 0,Y 587.181,Z 295.461,A -85,B 0,C 180,E1 -1544.557,E2 -1544.557} C_VEL
LIN {X 0,Y 587.206,Z 288.275,A -85,B 0,C 180,E1 -1547.41,E2 -1547.41} C_VEL
LIN {X 0,Y 587.214,Z 282.885,A -85,B 0,C 180,E1 -1549.579,E2 -1549.579} C_VEL
LIN {X 0,Y 587.252,Z 277.496,A -85,B 0,C 180,E1 -1551.777,E2 -1551.777} C_VEL
LIN {X 0,Y 587.296,Z 270.31,A -85,B 0,C 180,E1 -1554.761,E2 -1554.761} C_VEL
LIN {X 0,Y 587.302,Z 263.443,A -85,B 0,C 180,E1 -1557.682,E2 -1557.682} C_VEL
LIN {X 0,Y 587.337,Z 257.734,A -85,B 0,C 180,E1 -1560.169,E2 -1560.169} C_VEL
LIN {X 0,Y 587.372,Z 251.159,A -85,B 0,C 180,E1 -1563.115,E2 -1563.115} C_VEL
LIN {X 0,Y 587.375,Z 245.159,A -85,B 0,C 180,E1 -1565.893,E2 -1565.893} C_VEL
LIN {X 0,Y 587.429,Z 239.782,A -85,B 0,C 180,E1 -1568.471,E2 -1568.471} C_VEL
LIN {X 0,Y 587.532,Z 234.9,A -85,B 0,C 180,E1 -1571.139,E2 -1571.139} C_VEL
LIN {X 0,Y 587.374,Z 233.314,A -85,B 0,C 180,E1 -1572.11,E2 -1572.11} C_VEL
LIN {X 0,Y 587.294,Z 232.833,A -85,B 0,C 180,E1 -1573.114,E2 -1573.114} C_VEL
LIN {X 0,Y 587.303,Z 232.824,A -85,B 0,C 180,E1 -1576.045,E2 -1576.045} C_VEL
LIN {X 0,Y 587.313,Z 232.831,A -85,B 0,C 180,E1 -1578.926,E2 -1578.926} C_VEL
LIN {X 0,Y 587.306,Z 232.824,A -85,B 0,C 180,E1 -1581.516,E2 -1581.516} C_VEL
LIN {X 0,Y 587.278,Z 232.827,A -85,B 0,C 180,E1 -1584.097,E2 -1584.097} C_VEL
LIN {X 0,Y 587.334,Z 232.825,A -85,B 0,C 180,E1 -1586.887,E2 -1586.887} C_VEL
LIN {X 0,Y 587.317,Z 232.821,A -85,B 0,C 180,E1 -1589.492,E2 -1589.492} C_VEL
LIN {X 0,Y 587.289,Z 232.829,A -85,B 0,C 180,E1 -1592.177,E2 -1592.177} C_VEL
LIN {X 0,Y 587.328,Z 232.829,A -85,B 0,C 180,E1 -1594.48,E2 -1594.48} C_VEL
LIN {X 0,Y 587.305,Z 232.822,A -85,B 0,C 180,E1 -1597.482,E2 -1597.482} C_VEL
LIN {X 0,Y 587.305,Z 232.824,A -85,B 0,C 180,E1 -1599.691,E2 -1599.691} C_VEL
LIN {X 0,Y 587.281,Z 232.829,A -85,B 0,C 180,E1 -1601.869,E2 -1601.869} C_VEL
LIN {X 0,Y 587.3,Z 232.824,A -85,B 0,C 180,E1 -1604.733,E2 -1604.733} C_VEL
LIN {X 0,Y 587.289,Z 232.825,A -85,B 0,C 180,E1 -1606.854,E2 -1606.854} C_VEL
LIN {X 0,Y 587.323,Z 232.824,A -85,B 0,C 180,E1 -1609.656,E2 -1609.656} C_VEL
LIN {X 0,Y 587.305,Z 232.824,A -85,B 0,C 180,E1 -1612.433,E2 -1612.433} C_VEL
LIN {X 0,Y 587.339,Z 232.819,A -85,B 0,C 180,E1 -1615.192,E2 -1615.192} C_VEL
LIN {X 0,Y 587.347,Z 232.824,A -85,B 0,C 180,E1 -1617.939,E2 -1617.939} C_VEL
LIN {X 0,Y 587.36,Z 232.82,A -85,B 0,C 180,E1 -1619.996,E2 -1619.996} C_VEL
LIN {X 0,Y 587.336,Z 232.818,A -85,B 0,C 180,E1 -1622.739,E2 -1622.739} C_VEL
LIN {X 0,Y 587.342,Z 232.827,A -85,B 0,C 180,E1 -1625.489,E2 -1625.489} C_VEL
LIN {X 0,Y 587.302,Z 232.823,A -85,B 0,C 180,E1 -1628.252,E2 -1628.252} C_VEL
LIN {X 0,Y 587.365,Z 232.821,A -85,B 0,C 180,E1 -1631.146,E2 -1631.146} C_VEL
LIN {X 0,Y 587.288,Z 232.824,A -85,B 0,C 180,E1 -1634.234,E2 -1634.234} C_VEL
LIN {X 0,Y 587.323,Z 232.824,A -85,B 0,C 180,E1 -1636.809,E2 -1636.809} C_VEL
LIN {X 0,Y 587.273,Z 232.826,A -85,B 0,C 180,E1 -1638.272,E2 -1638.272} C_VEL
LIN {X 0,Y 586.636,Z 232.912,A -85,B 0,C 180,E1 -1638.844,E2 -1638.844} C_VEL
LIN {X 0,Y 583.825,Z 233.267,A -85,B 0,C 180,E1 -1639.773,E2 -1639.773} C_VEL
LIN {X 0,Y 581.418,Z 233.568,A -85,B 0,C 180,E1 -1640.52,E2 -1640.52} C_VEL
LIN {X 0,Y 580.357,Z 233.697,A -85,B 0,C 180,E1 -1641.097,E2 -1641.097} C_VEL
LIN {X 0,Y 580.257,Z 233.706,A -85,B 0,C 180,E1 -1641.292,E2 -1641.292} C_VEL
LIN {X 0,Y 580.241,Z 233.704,A -85,B 0,C 180,E1 -1643.554,E2 -1643.554} C_VEL
LIN {X 0,Y 580.245,Z 233.702,A -85,B 0,C 180,E1 -1645.845,E2 -1645.845} C_VEL
LIN {X 0,Y 580.268,Z 233.7,A -85,B 0,C 180,E1 -1648.181,E2 -1648.181} C_VEL
LIN {X 0,Y 580.248,Z 233.71,A -85,B 0,C 180,E1 -1650.69,E2 -1650.69} C_VEL
LIN {X 0,Y 580.261,Z 233.701,A -85,B 0,C 180,E1 -1653.312,E2 -1653.312} C_VEL
LIN {X 0,Y 580.285,Z 233.697,A -85,B 0,C 180,E1 -1655.763,E2 -1655.763} C_VEL
LIN {X 0,Y 580.245,Z 233.705,A -85,B 0,C 180,E1 -1658.142,E2 -1658.142} C_VEL
LIN {X 0,Y 580.255,Z 233.704,A -85,B 0,C 180,E1 -1660.839,E2 -1660.839} C_VEL
LIN {X 0,Y 580.242,Z 233.703,A -85,B 0,C 180,E1 -1663.652,E2 -1663.652} C_VEL
LIN {X 0,Y 580.233,Z 233.708,A -85,B 0,C 180,E1 -1666.604,E2 -1666.604} C_VEL
LIN {X 0,Y 580.267,Z 233.699,A -85,B 0,C 180,E1 -1669.155,E2 -1669.155} C_VEL
LIN {X 0,Y 580.24,Z 233.709,A -85,B 0,C 180,E1 -1671.922,E2 -1671.922} C_VEL
LIN {X 0,Y 580.252,Z 233.705,A -85,B 0,C 180,E1 -1674.453,E2 -1674.453} C_VEL
LIN {X 0,Y 580.239,Z 233.702,A -85,B 0,C 180,E1 -1676.973,E2 -1676.973} C_VEL
LIN {X 0,Y 580.268,Z 233.701,A -85,B 0,C 180,E1 -1679.424,E2 -1679.424} C_VEL
LIN {X 0,Y 580.259,Z 233.705,A -85,B 0,C 180,E1 -1682.133,E2 -1682.133} C_VEL
LIN {X 0,Y 580.255,Z 233.701,A -85,B 0,C 180,E1 -1684.918,E2 -1684.918} C_VEL
LIN {X 0,Y 580.29,Z 233.699,A -85,B 0,C 180,E1 -1687.198,E2 -1687.198} C_VEL
LIN {X 0,Y 580.254,Z 233.702,A -85,B 0,C 180,E1 -1690.176,E2 -1690.176} C_VEL
LIN {X 0,Y 580.28,Z 233.702,A -85,B 0,C 180,E1 -1693.102,E2 -1693.102} C_VEL
LIN {X 0,Y 580.268,Z 233.701,A -85,B 0,C 180,E1 -1695.982,E2 -1695.982} C_VEL
LIN {X 0,Y 580.28,Z 233.7,A -85,B 0,C 180,E1 -1698.827,E2 -1698.827} C_VEL
LIN {X 0,Y 580.282,Z 233.702,A -85,B 0,C 180,E1 -1701.643,E2 -1701.643} C_VEL
LIN {X 0,Y 580.231,Z 233.706,A -85,B 0,C 180,E1 -1703.742,E2 -1703.742} C_VEL
LIN {X 0,Y 580.211,Z 233.708,A -85,B 0,C 180,E1 -1705.832,E2 -1705.832} C_VEL
LIN {X 0,Y 580.268,Z 233.699,A -85,B 0,C 180,E1 -1707.918,E2 -1707.918} C_VEL
LIN {X 0,Y 580.314,Z 233.699,A -85,B 0,C 180,E1 -1710.694,E2 -1710.694} C_VEL
LIN {X 0,Y 580.237,Z 233.705,A -85,B 0,C 180,E1 -1713.472,E2 -1713.472} C_VEL
LIN {X 0,Y 580.269,Z 233.7,A -85,B 0,C 180,E1 -1715.56,E2 -1715.56} C_VEL
LIN {X 0,Y 580.274,Z 233.699,A -85,B 0,C 180,E1 -1717.656,E2 -1717.656} C_VEL
LIN {X 0,Y 580.253,Z 233.708,A -85,B 0,C 180,E1 -1720.467,E2 -1720.467} C_VEL
LIN {X 0,Y 580.24,Z 233.704,A -85,B 0,C 180,E1 -1723.305,E2 -1723.305} C_VEL
LIN {X 0,Y 580.24,Z 233.707,A -85,B 0,C 180,E1 -1726.175,E2 -1726.175} C_VEL
LIN {X 0,Y 580.268,Z 233.7,A -85,B 0,C 180,E1 -1729.087,E2 -1729.087} C_VEL
LIN {X 0,Y 580.238,Z 233.708,A -85,B 0,C 180,E1 -1732.054,E2 -1732.054} C_VEL
LIN {X 0,Y 580.275,Z 233.701,A -85,B 0,C 180,E1 -1734.737,E2 -1734.737} C_VEL
LIN {X 0,Y 580.23,Z 233.704,A -85,B 0,C 180,E1 -1737.404,E2 -1737.404} C_VEL
LIN {X 0,Y 580.254,Z 233.705,A -85,B 0,C 180,E1 -1739.774,E2 -1739.774} C_VEL
LIN {X 0,Y 580.249,Z 233.708,A -85,B 0,C 180,E1 -1742.203,E2 -1742.203} C_VEL
LIN {X 0,Y 580.246,Z 233.702,A -85,B 0,C 180,E1 -1744.699,E2 -1744.699} C_VEL
LIN {X 0,Y 580.246,Z 233.703,A -85,B 0,C 180,E1 -1747.272,E2 -1747.272} C_VEL
LIN {X 0,Y 580.256,Z 233.703,A -85,B 0,C 180,E1 -1750.277,E2 -1750.277} C_VEL
LIN {X 0,Y 580.228,Z 233.704,A -85,B 0,C 180,E1 -1752.71,E2 -1752.71} C_VEL
LIN {X 0,Y 580.223,Z 233.714,A -85,B 0,C 180,E1 -1755.613,E2 -1755.613} C_VEL
LIN {X 0,Y 580.266,Z 233.7,A -85,B 0,C 180,E1 -1758.239,E2 -1758.239} C_VEL
LIN {X 0,Y 580.235,Z 233.705,A -85,B 0,C 180,E1 -1760.97,E2 -1760.97} C_VEL
LIN {X 0,Y 580.255,Z 233.707,A -85,B 0,C 180,E1 -1763.603,E2 -1763.603} C_VEL
LIN {X 0,Y 580.268,Z 233.699,A -85,B 0,C 180,E1 -1766.149,E2 -1766.149} C_VEL
LIN {X 0,Y 580.239,Z 233.704,A -85,B 0,C 180,E1 -1768.619,E2 -1768.619} C_VEL
LIN {X 0,Y 580.261,Z 233.707,A -85,B 0,C 180,E1 -1771.029,E2 -1771.029} C_VEL
LIN {X 0,Y 580.256,Z 233.702,A -85,B 0,C 180,E1 -1773.671,E2 -1773.671} C_VEL
LIN {X 0,Y 580.263,Z 233.701,A -85,B 0,C 180,E1 -1775.688,E2 -1775.688} C_VEL
LIN {X 0,Y 580.239,Z 233.702,A -85,B 0,C 180,E1 -1777.952,E2 -1777.952} C_VEL
LIN {X 0,Y 580.272,Z 233.708,A -85,B 0,C 180,E1 -1780.918,E2 -1780.918} C_VEL
LIN {X 0,Y 580.245,Z 233.702,A -85,B 0,C 180,E1 -1783.83,E2 -1783.83} C_VEL
LIN {X 0,Y 580.244,Z 233.712,A -85,B 0,C 180,E1 -1786.7,E2 -1786.7} C_VEL
LIN {X 0,Y 580.335,Z 233.697,A -85,B 0,C 180,E1 -1788.832,E2 -1788.832} C_VEL
LIN {X 0,Y 580.276,Z 233.698,A -85,B 0,C 180,E1 -1791.648,E2 -1791.648} C_VEL
LIN {X 0,Y 580.305,Z 233.704,A -85,B 0,C 180,E1 -1794.444,E2 -1794.444} C_VEL
LIN {X 0,Y 580.305,Z 233.694,A -85,B 0,C 180,E1 -1797.228,E2 -1797.228} C_VEL
LIN {X 0,Y 580.33,Z 233.696,A -85,B 0,C 180,E1 -1800.004,E2 -1800.004} C_VEL
LIN {X 0,Y 580.317,Z 233.695,A -85,B 0,C 180,E1 -1802.781,E2 -1802.781} C_VEL
LIN {X 0,Y 580.289,Z 233.698,A -85,B 0,C 180,E1 -1805.564,E2 -1805.564} C_VEL
LIN {X 0,Y 580.299,Z 233.7,A -85,B 0,C 180,E1 -1808.36,E2 -1808.36} C_VEL
LIN {X 0,Y 580.298,Z 233.695,A -85,B 0,C 180,E1 -1811.195,E2 -1811.195} C_VEL
LIN {X 0,Y 580.308,Z 233.702,A -85,B 0,C 180,E1 -1814.021,E2 -1814.021} C_VEL
LIN {X 0,Y 580.231,Z 233.703,A -85,B 0,C 180,E1 -1816.903,E2 -1816.903} C_VEL
LIN {X 0,Y 580.272,Z 233.706,A -85,B 0,C 180,E1 -1819.826,E2 -1819.826} C_VEL
LIN {X 0,Y 580.278,Z 233.698,A -85,B 0,C 180,E1 -1822.806,E2 -1822.806} C_VEL
LIN {X 0,Y 580.264,Z 233.704,A -85,B 0,C 180,E1 -1825.853,E2 -1825.853} C_VEL
LIN {X 0,Y 580.278,Z 233.7,A -85,B 0,C 180,E1 -1828.98,E2 -1828.98} C_VEL
LIN {X 0,Y 580.269,Z 233.709,A -85,B 0,C 180,E1 -1831.388,E2 -1831.388} C_VEL
LIN {X 0,Y 580.275,Z 233.7,A -85,B 0,C 180,E1 -1833.86,E2 -1833.86} C_VEL
LIN {X 0,Y 580.278,Z 233.704,A -85,B 0,C 180,E1 -1836.933,E2 -1836.933} C_VEL
LIN {X 0,Y 580.272,Z 233.7,A -85,B 0,C 180,E1 -1839.937,E2 -1839.937} C_VEL
LIN {X 0,Y 580.255,Z 233.706,A -85,B 0,C 180,E1 -1842.711,E2 -1842.711} C_VEL
LIN {X 0,Y 580.255,Z 233.706,A -85,B 0,C 180,E1 -1845.613,E2 -1845.613} C_VEL
LIN {X 0,Y 580.241,Z 233.711,A -85,B 0,C 180,E1 -1847.291,E2 -1847.291} C_VEL
LIN {X 0,Y 580.535,Z 236.79,A -85,B 0,C 180,E1 -1849.178,E2 -1849.178} C_VEL
LIN {X 0,Y 580.437,Z 241.761,A -85,B 0,C 180,E1 -1851.911,E2 -1851.911} C_VEL
LIN {X 0,Y 580.377,Z 246.955,A -85,B 0,C 180,E1 -1854.462,E2 -1854.462} C_VEL
LIN {X 0,Y 580.328,Z 252.345,A -85,B 0,C 180,E1 -1856.978,E2 -1856.978} C_VEL
LIN {X 0,Y 580.308,Z 257.734,A -85,B 0,C 180,E1 -1859.426,E2 -1859.426} C_VEL
LIN {X 0,Y 580.248,Z 263.902,A -85,B 0,C 180,E1 -1862.153,E2 -1862.153} C_VEL
LIN {X 0,Y 580.232,Z 270.31,A -85,B 0,C 180,E1 -1864.917,E2 -1864.917} C_VEL
LIN {X 0,Y 580.198,Z 277.496,A -85,B 0,C 180,E1 -1867.945,E2 -1867.945} C_VEL
LIN {X 0,Y 580.168,Z 284.682,A -85,B 0,C 180,E1 -1870.909,E2 -1870.909} C_VEL
LIN {X 0,Y 580.11,Z 291.868,A -85,B 0,C 180,E1 -1873.821,E2 -1873.821} C_VEL
LIN {X 0,Y 580.075,Z 299.054,A -85,B 0,C 180,E1 -1876.692,E2 -1876.692} C_VEL
LIN {X 0,Y 580.075,Z 301.552,A -85,B 0,C 180,E1 -1877.67,E2 -1877.67} C_VEL
LIN {X 0,Y 580.792,Z 306.403,A -85,B 0,C 180,E1 -1877.775,E2 -1877.775} C_VEL
LIN {X 0,Y 580.711,Z 319.848,A -85,B 0,C 180,E1 -1878.127,E2 -1878.127} C_VEL
LIN {X 0,Y 580.615,Z 330.285,A -85,B 0,C 180,E1 -1878.515,E2 -1878.515} C_VEL
LIN {X 0,Y 580.507,Z 342.207,A -85,B 0,C 180,E1 -1879.096,E2 -1879.096} C_VEL
LIN {X 0,Y 580.446,Z 353.481,A -85,B 0,C 180,E1 -1879.801,E2 -1879.801} C_VEL
LIN {X 0,Y 580.353,Z 363.645,A -85,B 0,C 180,E1 -1880.591,E2 -1880.591} C_VEL
LIN {X 0,Y 580.27,Z 372.773,A -85,B 0,C 180,E1 -1881.468,E2 -1881.468} C_VEL
LIN {X 0,Y 580.201,Z 381.679,A -85,B 0,C 180,E1 -1882.518,E2 -1882.518} C_VEL
LIN {X 0,Y 580.11,Z 389.3,A -85,B 0,C 180,E1 -1883.642,E2 -1883.642} C_VEL
LIN {X 0,Y 580.086,Z 395.365,A -85,B 0,C 180,E1 -1884.787,E2 -1884.787} C_VEL
LIN {X 0,Y 580.105,Z 399.669,A -85,B 0,C 180,E1 -1885.832,E2 -1885.832} C_VEL
LIN {X 0,Y 580.123,Z 401.962,A -85,B 0,C 180,E1 -1886.527,E2 -1886.527} C_VEL
LIN {X 0,Y 580.043,Z 403.8,A -85,B 0,C 180,E1 -1887.222,E2 -1887.222} C_VEL
LIN {X 0,Y 580.047,Z 406.187,A -85,B 0,C 180,E1 -1888.611,E2 -1888.611} C_VEL
LIN {X 0,Y 580.04,Z 406.782,A -85,B 0,C 180,E1 -1889.306,E2 -1889.306} C_VEL
LIN {X 0,Y 580.037,Z 406.983,A -85,B 0,C 180,E1 -1890,E2 -1890} C_VEL
LIN {X 0,Y 580.04,Z 406.782,A -85,B 0,C 180,E1 -1890.694,E2 -1890.694} C_VEL
LIN {X 0,Y 580.047,Z 406.187,A -85,B 0,C 180,E1 -1891.389,E2 -1891.389} C_VEL
LIN {X 0,Y 580.043,Z 403.8,A -85,B 0,C 180,E1 -1892.778,E2 -1892.778} C_VEL
LIN {X 0,Y 580.11,Z 400.89,A -85,B 0,C 180,E1 -1893.821,E2 -1893.821} C_VEL
LIN {X 0,Y 580.053,Z 396.943,A -85,B 0,C 180,E1 -1894.865,E2 -1894.865} C_VEL
LIN {X 0,Y 580.162,Z 391.849,A -85,B 0,C 180,E1 -1895.91,E2 -1895.91} C_VEL
LIN {X 0,Y 580.159,Z 385.465,A -85,B 0,C 180,E1 -1896.958,E2 -1896.958} C_VEL
LIN {X 0,Y 580.243,Z 377.486,A -85,B 0,C 180,E1 -1898.007,E2 -1898.007} C_VEL
LIN {X 0,Y 580.305,Z 369.345,A -85,B 0,C 180,E1 -1898.883,E2 -1898.883} C_VEL
LIN {X 0,Y 580.371,Z 359.377,A -85,B 0,C 180,E1 -1899.76,E2 -1899.76} C_VEL
LIN {X 0,Y 580.445,Z 349.562,A -85,B 0,C 180,E1 -1900.464,E2 -1900.464} C_VEL
LIN {X 0,Y 580.525,Z 338.935,A -85,B 0,C 180,E1 -1901.08,E2 -1901.08} C_VEL
LIN {X 0,Y 580.643,Z 326.143,A -85,B 0,C 180,E1 -1901.652,E2 -1901.652} C_VEL
LIN {X 0,Y 580.771,Z 313.904,A -85,B 0,C 180,E1 -1902.049,E2 -1902.049} C_VEL
LIN {X 0,Y 580.55,Z 304.504,A -85,B 0,C 180,E1 -1902.267,E2 -1902.267} C_VEL
LIN {X 0,Y 580.078,Z 301.468,A -85,B 0,C 180,E1 -1902.352,E2 -1902.352} C_VEL
LIN {X 0,Y 580.107,Z 295.461,A -85,B 0,C 180,E1 -1904.739,E2 -1904.739} C_VEL
LIN {X 0,Y 580.136,Z 288.275,A -85,B 0,C 180,E1 -1907.629,E2 -1907.629} C_VEL
LIN {X 0,Y 580.159,Z 282.885,A -85,B 0,C 180,E1 -1909.827,E2 -1909.827} C_VEL
LIN {X 0,Y 580.201,Z 277.496,A -85,B 0,C 180,E1 -1912.055,E2 -1912.055} C_VEL
LIN {X 0,Y 580.232,Z 270.31,A -85,B 0,C 180,E1 -1915.083,E2 -1915.083} C_VEL
LIN {X 0,Y 580.248,Z 263.902,A -85,B 0,C 180,E1 -1917.847,E2 -1917.847} C_VEL
LIN {X 0,Y 580.3,Z 257.465,A -85,B 0,C 180,E1 -1920.695,E2 -1920.695} C_VEL
LIN {X 0,Y 580.344,Z 251.696,A -85,B 0,C 180,E1 -1923.32,E2 -1923.32} C_VEL
LIN {X 0,Y 580.376,Z 245.159,A -85,B 0,C 180,E1 -1926.395,E2 -1926.395} C_VEL
LIN {X 0,Y 580.48,Z 239.7,A -85,B 0,C 180,E1 -1929.205,E2 -1929.205} C_VEL
LIN {X 0,Y 580.514,Z 235.886,A -85,B 0,C 180,E1 -1931.355,E2 -1931.355} C_VEL
LIN {X 0,Y 580.241,Z 233.711,A -85,B 0,C 180,E1 -1932.709,E2 -1932.709} C_VEL
LIN {X 0,Y 580.255,Z 233.704,A -85,B 0,C 180,E1 -1935.61,E2 -1935.61} C_VEL
LIN {X 0,Y 580.244,Z 233.704,A -85,B 0,C 180,E1 -1938.226,E2 -1938.226} C_VEL
LIN {X 0,Y 580.264,Z 233.708,A -85,B 0,C 180,E1 -1940.962,E2 -1940.962} C_VEL
LIN {X 0,Y 580.245,Z 233.702,A -85,B 0,C 180,E1 -1943.592,E2 -1943.592} C_VEL
LIN {X 0,Y 580.275,Z 233.7,A -85,B 0,C 180,E1 -1946.14,E2 -1946.14} C_VEL
LIN {X 0,Y 580.269,Z 233.709,A -85,B 0,C 180,E1 -1948.612,E2 -1948.612} C_VEL
LIN {X 0,Y 580.278,Z 233.7,A -85,B 0,C 180,E1 -1951.02,E2 -1951.02} C_VEL
LIN {X 0,Y 580.264,Z 233.704,A -85,B 0,C 180,E1 -1954.147,E2 -1954.147} C_VEL
LIN {X 0,Y 580.278,Z 233.698,A -85,B 0,C 180,E1 -1957.194,E2 -1957.194} C_VEL
LIN {X 0,Y 580.272,Z 233.706,A -85,B 0,C 180,E1 -1960.174,E2 -1960.174} C_VEL
LIN {X 0,Y 580.232,Z 233.703,A -85,B 0,C 180,E1 -1963.109,E2 -1963.109} C_VEL
LIN {X 0,Y 580.308,Z 233.702,A -85,B 0,C 180,E1 -1965.979,E2 -1965.979} C_VEL
LIN {X 0,Y 580.303,Z 233.695,A -85,B 0,C 180,E1 -1968.823,E2 -1968.823} C_VEL
LIN {X 0,Y 580.299,Z 233.7,A -85,B 0,C 180,E1 -1971.64,E2 -1971.64} C_VEL
LIN {X 0,Y 580.289,Z 233.698,A -85,B 0,C 180,E1 -1974.436,E2 -1974.436} C_VEL
LIN {X 0,Y 580.317,Z 233.695,A -85,B 0,C 180,E1 -1977.219,E2 -1977.219} C_VEL
LIN {X 0,Y 580.33,Z 233.696,A -85,B 0,C 180,E1 -1979.996,E2 -1979.996} C_VEL
LIN {X 0,Y 580.305,Z 233.694,A -85,B 0,C 180,E1 -1982.772,E2 -1982.772} C_VEL
LIN {X 0,Y 580.305,Z 233.704,A -85,B 0,C 180,E1 -1985.556,E2 -1985.556} C_VEL
LIN {X 0,Y 580.276,Z 233.698,A -85,B 0,C 180,E1 -1988.352,E2 -1988.352} C_VEL
LIN {X 0,Y 580.317,Z 233.7,A -85,B 0,C 180,E1 -1991.204,E2 -1991.204} C_VEL
LIN {X 0,Y 580.252,Z 233.701,A -85,B 0,C 180,E1 -1994.318,E2 -1994.318} C_VEL
LIN {X 0,Y 580.289,Z 233.702,A -85,B 0,C 180,E1 -1996.909,E2 -1996.909} C_VEL
LIN {X 0,Y 580.258,Z 233.701,A -85,B 0,C 180,E1 -1999.818,E2 -1999.818} C_VEL
LIN {X 0,Y 580.257,Z 233.706,A -85,B 0,C 180,E1 -2001.292,E2 -2001.292} C_VEL
LIN {X 0,Y 579.547,Z 233.791,A -85,B 0,C 180,E1 -2001.871,E2 -2001.871} C_VEL
LIN {X 0,Y 576.666,Z 234.154,A -85,B 0,C 180,E1 -2002.811,E2 -2002.811} C_VEL
LIN {X 0,Y 574.276,Z 234.448,A -85,B 0,C 180,E1 -2003.567,E2 -2003.567} C_VEL
LIN {X 0,Y 573.279,Z 234.57,A -85,B 0,C 180,E1 -2004.151,E2 -2004.151} C_VEL
LIN {X 0,Y 573.213,Z 234.579,A -85,B 0,C 180,E1 -2004.349,E2 -2004.349} C_VEL
LIN {X 0,Y 573.218,Z 234.585,A -85,B 0,C 180,E1 -2006.971,E2 -2006.971} C_VEL
LIN {X 0,Y 573.211,Z 234.579,A -85,B 0,C 180,E1 -2009.484,E2 -2009.484} C_VEL
LIN {X 0,Y 573.216,Z 234.586,A -85,B 0,C 180,E1 -2012.64,E2 -2012.64} C_VEL
LIN {X 0,Y 573.228,Z 234.578,A -85,B 0,C 180,E1 -2015.179,E2 -2015.179} C_VEL
LIN {X 0,Y 573.193,Z 234.581,A -85,B 0,C 180,E1 -2017.803,E2 -2017.803} C_VEL
LIN {X 0,Y 573.223,Z 234.586,A -85,B 0,C 180,E1 -2020.524,E2 -2020.524} C_VEL
LIN {X 0,Y 573.207,Z 234.578,A -85,B 0,C 180,E1 -2023.353,E2 -2023.353} C_VEL
LIN {X 0,Y 573.201,Z 234.589,A -85,B 0,C 180,E1 -2026.326,E2 -2026.326} C_VEL
LIN {X 0,Y 573.219,Z 234.577,A -85,B 0,C 180,E1 -2029.474,E2 -2029.474} C_VEL
LIN {X 0,Y 573.185,Z 234.59,A -85,B 0,C 180,E1 -2032.189,E2 -2032.189} C_VEL
LIN {X 0,Y 573.213,Z 234.578,A -85,B 0,C 180,E1 -2034.813,E2 -2034.813} C_VEL
LIN {X 0,Y 573.202,Z 234.58,A -85,B 0,C 180,E1 -2037.352,E2 -2037.352} C_VEL
LIN {X 0,Y 573.224,Z 234.578,A -85,B 0,C 180,E1 -2040.501,E2 -2040.501} C_VEL
LIN {X 0,Y 573.206,Z 234.579,A -85,B 0,C 180,E1 -2043.022,E2 -2043.022} C_VEL
LIN {X 0,Y 573.229,Z 234.58,A -85,B 0,C 180,E1 -2045.364,E2 -2045.364} C_VEL
LIN {X 0,Y 573.21,Z 234.588,A -85,B 0,C 180,E1 -2047.662,E2 -2047.662} C_VEL
LIN {X 0,Y 573.212,Z 234.578,A -85,B 0,C 180,E1 -2050.725,E2 -2050.725} C_VEL
LIN {X 0,Y 573.213,Z 234.586,A -85,B 0,C 180,E1 -2053.621,E2 -2053.621} C_VEL
LIN {X 0,Y 573.194,Z 234.581,A -85,B 0,C 180,E1 -2056.529,E2 -2056.529} C_VEL
LIN {X 0,Y 573.222,Z 234.586,A -85,B 0,C 180,E1 -2059.403,E2 -2059.403} C_VEL
LIN {X 0,Y 573.225,Z 234.577,A -85,B 0,C 180,E1 -2062.249,E2 -2062.249} C_VEL
LIN {X 0,Y 573.235,Z 234.576,A -85,B 0,C 180,E1 -2064.371,E2 -2064.371} C_VEL
LIN {X 0,Y 573.258,Z 234.581,A -85,B 0,C 180,E1 -2067.189,E2 -2067.189} C_VEL
LIN {X 0,Y 573.248,Z 234.574,A -85,B 0,C 180,E1 -2070,E2 -2070} C_VEL
LIN {X 0,Y 573.258,Z 234.581,A -85,B 0,C 180,E1 -2072.811,E2 -2072.811} C_VEL
LIN {X 0,Y 573.235,Z 234.576,A -85,B 0,C 180,E1 -2075.629,E2 -2075.629} C_VEL
LIN {X 0,Y 573.225,Z 234.577,A -85,B 0,C 180,E1 -2077.751,E2 -2077.751} C_VEL
LIN {X 0,Y 573.222,Z 234.586,A -85,B 0,C 180,E1 -2080.597,E2 -2080.597} C_VEL
LIN {X 0,Y 573.194,Z 234.581,A -85,B 0,C 180,E1 -2083.471,E2 -2083.471} C_VEL
LIN {X 0,Y 573.213,Z 234.586,A -85,B 0,C 180,E1 -2086.379,E2 -2086.379} C_VEL
LIN {X 0,Y 573.209,Z 234.578,A -85,B 0,C 180,E1 -2089.332,E2 -2089.332} C_VEL
LIN {X 0,Y 573.21,Z 234.588,A -85,B 0,C 180,E1 -2092.338,E2 -2092.338} C_VEL
LIN {X 0,Y 573.219,Z 234.578,A -85,B 0,C 180,E1 -2094.885,E2 -2094.885} C_VEL
LIN {X 0,Y 573.228,Z 234.579,A -85,B 0,C 180,E1 -2097.768,E2 -2097.768} C_VEL
LIN {X 0,Y 573.213,Z 234.586,A -85,B 0,C 180,E1 -2100.177,E2 -2100.177} C_VEL
LIN {X 0,Y 573.202,Z 234.58,A -85,B 0,C 180,E1 -2102.648,E2 -2102.648} C_VEL
LIN {X 0,Y 573.213,Z 234.578,A -85,B 0,C 180,E1 -2105.187,E2 -2105.187} C_VEL
LIN {X 0,Y 573.185,Z 234.59,A -85,B 0,C 180,E1 -2107.811,E2 -2107.811} C_VEL
LIN {X 0,Y 573.215,Z 234.578,A -85,B 0,C 180,E1 -2110.532,E2 -2110.532} C_VEL
LIN {X 0,Y 573.201,Z 234.589,A -85,B 0,C 180,E1 -2113.674,E2 -2113.674} C_VEL
LIN {X 0,Y 573.207,Z 234.578,A -85,B 0,C 180,E1 -2116.647,E2 -2116.647} C_VEL
LIN {X 0,Y 573.228,Z 234.585,A -85,B 0,C 180,E1 -2119.482,E2 -2119.482} C_VEL
LIN {X 0,Y 573.193,Z 234.581,A -85,B 0,C 180,E1 -2122.197,E2 -2122.197} C_VEL
LIN {X 0,Y 573.228,Z 234.578,A -85,B 0,C 180,E1 -2124.821,E2 -2124.821} C_VEL
LIN {X 0,Y 573.215,Z 234.58,A -85,B 0,C 180,E1 -2127.776,E2 -2127.776} C_VEL
LIN {X 0,Y 573.23,Z 234.578,A -85,B 0,C 180,E1 -2130.639,E2 -2130.639} C_VEL
LIN {X 0,Y 573.218,Z 234.585,A -85,B 0,C 180,E1 -2133.029,E2 -2133.029} C_VEL
LIN {X 0,Y 573.242,Z 234.579,A -85,B 0,C 180,E1 -2135.371,E2 -2135.371} C_VEL
LIN {X 0,Y 573.199,Z 234.581,A -85,B 0,C 180,E1 -2138.424,E2 -2138.424} C_VEL
LIN {X 0,Y 573.243,Z 234.581,A -85,B 0,C 180,E1 -2140.736,E2 -2140.736} C_VEL
LIN {X 0,Y 573.219,Z 234.577,A -85,B 0,C 180,E1 -2143.626,E2 -2143.626} C_VEL
LIN {X 0,Y 573.197,Z 234.586,A -85,B 0,C 180,E1 -2146.534,E2 -2146.534} C_VEL
LIN {X 0,Y 573.266,Z 234.579,A -85,B 0,C 180,E1 -2148.739,E2 -2148.739} C_VEL
LIN {X 0,Y 573.223,Z 234.576,A -85,B 0,C 180,E1 -2151.544,E2 -2151.544} C_VEL
LIN {X 0,Y 573.199,Z 234.58,A -85,B 0,C 180,E1 -2153.669,E2 -2153.669} C_VEL
LIN {X 0,Y 573.192,Z 234.581,A -85,B 0,C 180,E1 -2155.785,E2 -2155.785} C_VEL
LIN {X 0,Y 573.283,Z 234.572,A -85,B 0,C 180,E1 -2157.897,E2 -2157.897} C_VEL
LIN {X 0,Y 573.319,Z 234.568,A -85,B 0,C 180,E1 -2160.706,E2 -2160.706} C_VEL
LIN {X 0,Y 573.282,Z 234.571,A -85,B 0,C 180,E1 -2162.815,E2 -2162.815} C_VEL
LIN {X 0,Y 573.258,Z 234.574,A -85,B 0,C 180,E1 -2165.632,E2 -2165.632} C_VEL
LIN {X 0,Y 573.242,Z 234.578,A -85,B 0,C 180,E1 -2168.464,E2 -2168.464} C_VEL
LIN {X 0,Y 573.269,Z 234.572,A -85,B 0,C 180,E1 -2171.315,E2 -2171.315} C_VEL
LIN {X 0,Y 573.269,Z 234.573,A -85,B 0,C 180,E1 -2174.423,E2 -2174.423} C_VEL
LIN {X 0,Y 573.18,Z 234.583,A -85,B 0,C 180,E1 -2177.117,E2 -2177.117} C_VEL
LIN {X 0,Y 573.266,Z 234.575,A -85,B 0,C 180,E1 -2179.333,E2 -2179.333} C_VEL
LIN {X 0,Y 573.217,Z 234.578,A -85,B 0,C 180,E1 -2182.342,E2 -2182.342} C_VEL
LIN {X 0,Y 573.233,Z 234.583,A -85,B 0,C 180,E1 -2185.414,E2 -2185.414} C_VEL
LIN {X 0,Y 573.198,Z 234.58,A -85,B 0,C 180,E1 -2188.569,E2 -2188.569} C_VEL
LIN {X 0,Y 573.219,Z 234.581,A -85,B 0,C 180,E1 -2190.996,E2 -2190.996} C_VEL
LIN {X 0,Y 573.246,Z 234.581,A -85,B 0,C 180,E1 -2193.523,E2 -2193.523} C_VEL
LIN {X 0,Y 573.19,Z 234.582,A -85,B 0,C 180,E1 -2196.056,E2 -2196.056} C_VEL
LIN {X 0,Y 573.232,Z 234.579,A -85,B 0,C 180,E1 -2198.705,E2 -2198.705} C_VEL
LIN {X 0,Y 573.217,Z 234.583,A -85,B 0,C 180,E1 -2201.461,E2 -2201.461} C_VEL
LIN {X 0,Y 573.222,Z 234.581,A -85,B 0,C 180,E1 -2204.337,E2 -2204.337} C_VEL
LIN {X 0,Y 573.205,Z 234.587,A -85,B 0,C 180,E1 -2206.639,E2 -2206.639} C_VEL
LIN {X 0,Y 573.372,Z 235.539,A -85,B 0,C 180,E1 -2207.613,E2 -2207.613} C_VEL
LIN {X 0,Y 573.551,Z 238.678,A -85,B 0,C 180,E1 -2209.502,E2 -2209.502} C_VEL
LIN {X 0,Y 573.412,Z 243.573,A -85,B 0,C 180,E1 -2212.207,E2 -2212.207} C_VEL
LIN {X 0,Y 573.319,Z 248.752,A -85,B 0,C 180,E1 -2214.821,E2 -2214.821} C_VEL
LIN {X 0,Y 573.276,Z 254.141,A -85,B 0,C 180,E1 -2217.357,E2 -2217.357} C_VEL
LIN {X 0,Y 573.25,Z 259.531,A -85,B 0,C 180,E1 -2219.825,E2 -2219.825} C_VEL
LIN {X 0,Y 573.192,Z 264.92,A -85,B 0,C 180,E1 -2222.231,E2 -2222.231} C_VEL
LIN {X 0,Y 573.177,Z 271.599,A -85,B 0,C 180,E1 -2225.144,E2 -2225.144} C_VEL
LIN {X 0,Y 573.114,Z 277.496,A -85,B 0,C 180,E1 -2227.658,E2 -2227.658} C_VEL
LIN {X 0,Y 573.079,Z 282.885,A -85,B 0,C 180,E1 -2229.917,E2 -2229.917} C_VEL
LIN {X 0,Y 573.054,Z 290.071,A -85,B 0,C 180,E1 -2232.882,E2 -2232.882} C_VEL
LIN {X 0,Y 573.039,Z 297.257,A -85,B 0,C 180,E1 -2235.801,E2 -2235.801} C_VEL
LIN {X 0,Y 572.988,Z 301.525,A -85,B 0,C 180,E1 -2237.515,E2 -2237.515} C_VEL
LIN {X 0,Y 573.847,Z 307.537,A -85,B 0,C 180,E1 -2237.647,E2 -2237.647} C_VEL
LIN {X 0,Y 573.763,Z 319.841,A -85,B 0,C 180,E1 -2237.981,E2 -2237.981} C_VEL
LIN {X 0,Y 573.641,Z 331.367,A -85,B 0,C 180,E1 -2238.422,E2 -2238.422} C_VEL
LIN {X 0,Y 573.51,Z 342.577,A -85,B 0,C 180,E1 -2238.982,E2 -2238.982} C_VEL
LIN {X 0,Y 573.446,Z 354.75,A -85,B 0,C 180,E1 -2239.764,E2 -2239.764} C_VEL
LIN {X 0,Y 573.308,Z 363.644,A -85,B 0,C 180,E1 -2240.474,E2 -2240.474} C_VEL
LIN {X 0,Y 573.207,Z 372.769,A -85,B 0,C 180,E1 -2241.362,E2 -2241.362} C_VEL
LIN {X 0,Y 573.162,Z 380.317,A -85,B 0,C 180,E1 -2242.248,E2 -2242.248} C_VEL
LIN {X 0,Y 573.067,Z 387.71,A -85,B 0,C 180,E1 -2243.306,E2 -2243.306} C_VEL
LIN {X 0,Y 573.069,Z 393.682,A -85,B 0,C 180,E1 -2244.37,E2 -2244.37} C_VEL
LIN {X 0,Y 573.029,Z 398.377,A -85,B 0,C 180,E1 -2245.428,E2 -2245.428} C_VEL
LIN {X 0,Y 573.023,Z 401.963,A -85,B 0,C 180,E1 -2246.484,E2 -2246.484} C_VEL
LIN {X 0,Y 572.959,Z 403.797,A -85,B 0,C 180,E1 -2247.188,E2 -2247.188} C_VEL
LIN {X 0,Y 572.946,Z 406.188,A -85,B 0,C 180,E1 -2248.594,E2 -2248.594} C_VEL
LIN {X 0,Y 572.941,Z 406.782,A -85,B 0,C 180,E1 -2249.297,E2 -2249.297} C_VEL
LIN {X 0,Y 572.938,Z 406.979,A -85,B 0,C 180,E1 -2250,E2 -2250} C_VEL
LIN {X 0,Y 572.941,Z 406.782,A -85,B 0,C 180,E1 -2250.703,E2 -2250.703} C_VEL
LIN {X 0,Y 572.946,Z 406.188,A -85,B 0,C 180,E1 -2251.406,E2 -2251.406} C_VEL
LIN {X 0,Y 572.959,Z 403.797,A -85,B 0,C 180,E1 -2252.812,E2 -2252.812} C_VEL
LIN {X 0,Y 573.015,Z 400.887,A -85,B 0,C 180,E1 -2253.868,E2 -2253.868} C_VEL
LIN {X 0,Y 572.963,Z 396.939,A -85,B 0,C 180,E1 -2254.926,E2 -2254.926} C_VEL
LIN {X 0,Y 573.074,Z 391.844,A -85,B 0,C 180,E1 -2255.983,E2 -2255.983} C_VEL
LIN {X 0,Y 573.085,Z 385.461,A -85,B 0,C 180,E1 -2257.044,E2 -2257.044} C_VEL
LIN {X 0,Y 573.179,Z 377.487,A -85,B 0,C 180,E1 -2258.106,E2 -2258.106} C_VEL
LIN {X 0,Y 573.255,Z 369.347,A -85,B 0,C 180,E1 -2258.993,E2 -2258.993} C_VEL
LIN {X 0,Y 573.344,Z 359.371,A -85,B 0,C 180,E1 -2259.881,E2 -2259.881} C_VEL
LIN {X 0,Y 573.456,Z 349.555,A -85,B 0,C 180,E1 -2260.593,E2 -2260.593} C_VEL
LIN {X 0,Y 573.557,Z 338.767,A -85,B 0,C 180,E1 -2261.225,E2 -2261.225} C_VEL
LIN {X 0,Y 573.684,Z 326.146,A -85,B 0,C 180,E1 -2261.796,E2 -2261.796} C_VEL
LIN {X 0,Y 573.822,Z 313.888,A -85,B 0,C 180,E1 -2262.197,E2 -2262.197} C_VEL
LIN {X 0,Y 573.653,Z 305.552,A -85,B 0,C 180,E1 -2262.397,E2 -2262.397} C_VEL
LIN {X 0,Y 572.989,Z 301.525,A -85,B 0,C 180,E1 -2262.485,E2 -2262.485} C_VEL
LIN {X 0,Y 573.037,Z 295.461,A -85,B 0,C 180,E1 -2264.925,E2 -2264.925} C_VEL
LIN {X 0,Y 573.056,Z 288.275,A -85,B 0,C 180,E1 -2267.854,E2 -2267.854} C_VEL
LIN {X 0,Y 573.124,Z 281.089,A -85,B 0,C 180,E1 -2270.831,E2 -2270.831} C_VEL
LIN {X 0,Y 573.123,Z 273.903,A -85,B 0,C 180,E1 -2273.87,E2 -2273.87} C_VEL
LIN {X 0,Y 573.176,Z 267.861,A -85,B 0,C 180,E1 -2276.478,E2 -2276.478} C_VEL
LIN {X 0,Y 573.234,Z 261.067,A -85,B 0,C 180,E1 -2279.484,E2 -2279.484} C_VEL
LIN {X 0,Y 573.269,Z 255.036,A -85,B 0,C 180,E1 -2282.229,E2 -2282.229} C_VEL
LIN {X 0,Y 573.308,Z 249.591,A -85,B 0,C 180,E1 -2284.78,E2 -2284.78} C_VEL
LIN {X 0,Y 573.383,Z 244.712,A -85,B 0,C 180,E1 -2287.181,E2 -2287.181} C_VEL
LIN {X 0,Y 573.501,Z 240.304,A -85,B 0,C 180,E1 -2289.585,E2 -2289.585} C_VEL
LIN {X 0,Y 573.522,Z 236.77,A -85,B 0,C 180,E1 -2291.623,E2 -2291.623} C_VEL
LIN {X 0,Y 573.288,Z 235.136,A -85,B 0,C 180,E1 -2292.644,E2 -2292.644} C_VEL
LIN {X 0,Y 573.209,Z 234.584,A -85,B 0,C 180,E1 -2293.663,E2 -2293.663} C_VEL
LIN {X 0,Y 573.204,Z 234.585,A -85,B 0,C 180,E1 -2296.635,E2 -2296.635} C_VEL
LIN {X 0,Y 573.233,Z 234.578,A -85,B 0,C 180,E1 -2299.475,E2 -2299.475} C_VEL
LIN {X 0,Y 573.225,Z 234.579,A -85,B 0,C 180,E1 -2302.189,E2 -2302.189} C_VEL
LIN {X 0,Y 573.223,Z 234.579,A -85,B 0,C 180,E1 -2305.229,E2 -2305.229} C_VEL
LIN {X 0,Y 573.239,Z 234.575,A -85,B 0,C 180,E1 -2307.772,E2 -2307.772} C_VEL
LIN {X 0,Y 573.24,Z 234.583,A -85,B 0,C 180,E1 -2310.63,E2 -2310.63} C_VEL
LIN {X 0,Y 573.207,Z 234.578,A -85,B 0,C 180,E1 -2313.512,E2 -2313.512} C_VEL
LIN {X 0,Y 573.201,Z 234.585,A -85,B 0,C 180,E1 -2316.13,E2 -2316.13} C_VEL
LIN {X 0,Y 573.236,Z 234.579,A -85,B 0,C 180,E1 -2318.711,E2 -2318.711} C_VEL
LIN {X 0,Y 573.196,Z 234.58,A -85,B 0,C 180,E1 -2321.407,E2 -2321.407} C_VEL
LIN {X 0,Y 573.206,Z 234.585,A -85,B 0,C 180,E1 -2324.348,E2 -2324.348} C_VEL
LIN {X 0,Y 573.211,Z 234.581,A -85,B 0,C 180,E1 -2326.526,E2 -2326.526} C_VEL
LIN {X 0,Y 573.254,Z 234.574,A -85,B 0,C 180,E1 -2329.4,E2 -2329.4} C_VEL
LIN {X 0,Y 573.215,Z 234.582,A -85,B 0,C 180,E1 -2332.245,E2 -2332.245} C_VEL
LIN {X 0,Y 573.283,Z 234.569,A -85,B 0,C 180,E1 -2335.073,E2 -2335.073} C_VEL
LIN {X 0,Y 573.29,Z 234.576,A -85,B 0,C 180,E1 -2337.888,E2 -2337.888} C_VEL
LIN {X 0,Y 573.299,Z 234.572,A -85,B 0,C 180,E1 -2339.996,E2 -2339.996} C_VEL
LIN {X 0,Y 573.275,Z 234.57,A -85,B 0,C 180,E1 -2342.807,E2 -2342.807} C_VEL
LIN {X 0,Y 573.27,Z 234.579,A -85,B 0,C 180,E1 -2345.624,E2 -2345.624} C_VEL
LIN {X 0,Y 573.247,Z 234.578,A -85,B 0,C 180,E1 -2347.746,E2 -2347.746} C_VEL
LIN {X 0,Y 573.241,Z 234.575,A -85,B 0,C 180,E1 -2350.592,E2 -2350.592} C_VEL
LIN {X 0,Y 573.215,Z 234.579,A -85,B 0,C 180,E1 -2352.745,E2 -2352.745} C_VEL
LIN {X 0,Y 573.205,Z 234.582,A -85,B 0,C 180,E1 -2355.644,E2 -2355.644} C_VEL
LIN {X 0,Y 573.212,Z 234.579,A -85,B 0,C 180,E1 -2357.844,E2 -2357.844} C_VEL
LIN {X 0,Y 573.213,Z 234.578,A -85,B 0,C 180,E1 -2360.072,E2 -2360.072} C_VEL
LIN {X 0,Y 573.205,Z 234.58,A -85,B 0,C 180,E1 -2362.333,E2 -2362.333} C_VEL
LIN {X 0,Y 573.213,Z 234.579,A -85,B 0,C 180,E1 -2364.349,E2 -2364.349} C_VEL
LIN {X 0,Y 572.585,Z 234.666,A -85,B 0,C 180,E1 -2364.935,E2 -2364.935} C_VEL
LIN {X 0,Y 569.742,Z 235.019,A -85,B 0,C 180,E1 -2365.886,E2 -2365.886} C_VEL
LIN {X 0,Y 567.312,Z 235.32,A -85,B 0,C 180,E1 -2366.652,E2 -2366.652} C_VEL
LIN {X 0,Y 566.262,Z 235.448,A -85,B 0,C 180,E1 -2367.243,E2 -2367.243} C_VEL
LIN {X 0,Y 566.174,Z 235.456,A -85,B 0,C 180,E1 -2367.443,E2 -2367.443} C_VEL
LIN {X 0,Y 566.165,Z 235.456,A -85,B 0,C 180,E1 -2369.764,E2 -2369.764} C_VEL
LIN {X 0,Y 566.167,Z 235.46,A -85,B 0,C 180,E1 -2372.426,E2 -2372.426} C_VEL
LIN {X 0,Y 566.174,Z 235.459,A -85,B 0,C 180,E1 -2374.99,E2 -2374.99} C_VEL
LIN {X 0,Y 566.154,Z 235.457,A -85,B 0,C 180,E1 -2377.456,E2 -2377.456} C_VEL
LIN {X 0,Y 566.18,Z 235.459,A -85,B 0,C 180,E1 -2380.193,E2 -2380.193} C_VEL
LIN {X 0,Y 566.166,Z 235.457,A -85,B 0,C 180,E1 -2383.049,E2 -2383.049} C_VEL
LIN {X 0,Y 566.151,Z 235.463,A -85,B 0,C 180,E1 -2386.044,E2 -2386.044} C_VEL
LIN {X 0,Y 566.168,Z 235.457,A -85,B 0,C 180,E1 -2388.861,E2 -2388.861} C_VEL
LIN {X 0,Y 566.139,Z 235.461,A -85,B 0,C 180,E1 -2391.634,E2 -2391.634} C_VEL
LIN {X 0,Y 566.156,Z 235.462,A -85,B 0,C 180,E1 -2394.308,E2 -2394.308} C_VEL
LIN {X 0,Y 566.171,Z 235.455,A -85,B 0,C 180,E1 -2396.895,E2 -2396.895} C_VEL
LIN {X 0,Y 566.148,Z 235.46,A -85,B 0,C 180,E1 -2399.406,E2 -2399.406} C_VEL
LIN {X 0,Y 566.165,Z 235.465,A -85,B 0,C 180,E1 -2401.855,E2 -2401.855} C_VEL
LIN {X 0,Y 566.167,Z 235.458,A -85,B 0,C 180,E1 -2404.249,E2 -2404.249} C_VEL
LIN {X 0,Y 566.189,Z 235.453,A -85,B 0,C 180,E1 -2406.696,E2 -2406.696} C_VEL
LIN {X 0,Y 566.164,Z 235.465,A -85,B 0,C 180,E1 -2409.661,E2 -2409.661} C_VEL
LIN {X 0,Y 566.194,Z 235.453,A -85,B 0,C 180,E1 -2412.669,E2 -2412.669} C_VEL
LIN {X 0,Y 566.174,Z 235.462,A -85,B 0,C 180,E1 -2415.626,E2 -2415.626} C_VEL
LIN {X 0,Y 566.205,Z 235.452,A -85,B 0,C 180,E1 -2418.652,E2 -2418.652} C_VEL
LIN {X 0,Y 566.199,Z 235.459,A -85,B 0,C 180,E1 -2421.434,E2 -2421.434} C_VEL
LIN {X 0,Y 566.16,Z 235.461,A -85,B 0,C 180,E1 -2423.586,E2 -2423.586} C_VEL
LIN {X 0,Y 566.128,Z 235.463,A -85,B 0,C 180,E1 -2425.728,E2 -2425.728} C_VEL
LIN {X 0,Y 566.211,Z 235.451,A -85,B 0,C 180,E1 -2427.866,E2 -2427.866} C_VEL
LIN {X 0,Y 566.251,Z 235.452,A -85,B 0,C 180,E1 -2430.711,E2 -2430.711} C_VEL
LIN {X 0,Y 566.139,Z 235.461,A -85,B 0,C 180,E1 -2433.559,E2 -2433.559} C_VEL
LIN {X 0,Y 566.203,Z 235.452,A -85,B 0,C 180,E1 -2435.699,E2 -2435.699} C_VEL
LIN {X 0,Y 566.181,Z 235.455,A -85,B 0,C 180,E1 -2437.848,E2 -2437.848} C_VEL
LIN {X 0,Y 566.191,Z 235.462,A -85,B 0,C 180,E1 -2440.73,E2 -2440.73} C_VEL
LIN {X 0,Y 566.152,Z 235.458,A -85,B 0,C 180,E1 -2443.642,E2 -2443.642} C_VEL
LIN {X 0,Y 566.181,Z 235.463,A -85,B 0,C 180,E1 -2446.588,E2 -2446.588} C_VEL
LIN {X 0,Y 566.152,Z 235.457,A -85,B 0,C 180,E1 -2449.582,E2 -2449.582} C_VEL
LIN {X 0,Y 566.165,Z 235.46,A -85,B 0,C 180,E1 -2452.632,E2 -2452.632} C_VEL
LIN {X 0,Y 566.186,Z 235.453,A -85,B 0,C 180,E1 -2455.04,E2 -2455.04} C_VEL
LIN {X 0,Y 566.165,Z 235.456,A -85,B 0,C 180,E1 -2457.341,E2 -2457.341} C_VEL
LIN {X 0,Y 566.18,Z 235.458,A -85,B 0,C 180,E1 -2459.769,E2 -2459.769} C_VEL
LIN {X 0,Y 566.153,Z 235.461,A -85,B 0,C 180,E1 -2462.435,E2 -2462.435} C_VEL
LIN {X 0,Y 566.157,Z 235.456,A -85,B 0,C 180,E1 -2464.998,E2 -2464.998} C_VEL
LIN {X 0,Y 566.142,Z 235.462,A -85,B 0,C 180,E1 -2467.464,E2 -2467.464} C_VEL
LIN {X 0,Y 566.174,Z 235.458,A -85,B 0,C 180,E1 -2470.201,E2 -2470.201} C_VEL
LIN {X 0,Y 566.153,Z 235.458,A -85,B 0,C 180,E1 -2473.058,E2 -2473.058} C_VEL
LIN {X 0,Y 566.154,Z 235.46,A -85,B 0,C 180,E1 -2476.052,E2 -2476.052} C_VEL
LIN {X 0,Y 566.165,Z 235.457,A -85,B 0,C 180,E1 -2478.868,E2 -2478.868} C_VEL
LIN {X 0,Y 566.144,Z 235.465,A -85,B 0,C 180,E1 -2481.642,E2 -2481.642} C_VEL
LIN {X 0,Y 566.172,Z 235.455,A -85,B 0,C 180,E1 -2484.316,E2 -2484.316} C_VEL
LIN {X 0,Y 566.173,Z 235.458,A -85,B 0,C 180,E1 -2486.902,E2 -2486.902} C_VEL
LIN {X 0,Y 566.145,Z 235.465,A -85,B 0,C 180,E1 -2489.412,E2 -2489.412} C_VEL
LIN {X 0,Y 566.195,Z 235.453,A -85,B 0,C 180,E1 -2491.863,E2 -2491.863} C_VEL
LIN {X 0,Y 566.206,Z 235.46,A -85,B 0,C 180,E1 -2495.044,E2 -2495.044} C_VEL
LIN {X 0,Y 566.164,Z 235.456,A -85,B 0,C 180,E1 -2498.142,E2 -2498.142} C_VEL
LIN {X 0,Y 566.204,Z 235.456,A -85,B 0,C 180,E1 -2500.619,E2 -2500.619} C_VEL
LIN {X 0,Y 566.186,Z 235.454,A -85,B 0,C 180,E1 -2503.417,E2 -2503.417} C_VEL
LIN {X 0,Y 566.156,Z 235.461,A -85,B 0,C 180,E1 -2506.363,E2 -2506.363} C_VEL
LIN {X 0,Y 566.225,Z 235.458,A -85,B 0,C 180,E1 -2508.676,E2 -2508.676} C_VEL
LIN {X 0,Y 566.177,Z 235.454,A -85,B 0,C 180,E1 -2511.438,E2 -2511.438} C_VEL
LIN {X 0,Y 566.236,Z 235.454,A -85,B 0,C 180,E1 -2514.306,E2 -2514.306} C_VEL
LIN {X 0,Y 566.255,Z 235.447,A -85,B 0,C 180,E1 -2517.87,E2 -2517.87} C_VEL
LIN {X 0,Y 566.289,Z 235.443,A -85,B 0,C 180,E1 -2520.715,E2 -2520.715} C_VEL
LIN {X 0,Y 566.247,Z 235.447,A -85,B 0,C 180,E1 -2522.85,E2 -2522.85} C_VEL
LIN {X 0,Y 566.228,Z 235.451,A -85,B 0,C 180,E1 -2525.702,E2 -2525.702} C_VEL
LIN {X 0,Y 566.192,Z 235.455,A -85,B 0,C 180,E1 -2528.57,E2 -2528.57} C_VEL
LIN {X 0,Y 566.237,Z 235.449,A -85,B 0,C 180,E1 -2531.458,E2 -2531.458} C_VEL
LIN {X 0,Y 566.223,Z 235.45,A -85,B 0,C 180,E1 -2534.506,E2 -2534.506} C_VEL
LIN {X 0,Y 566.152,Z 235.46,A -85,B 0,C 180,E1 -2537.336,E2 -2537.336} C_VEL
LIN {X 0,Y 566.197,Z 235.459,A -85,B 0,C 180,E1 -2539.584,E2 -2539.584} C_VEL
LIN {X 0,Y 566.183,Z 235.46,A -85,B 0,C 180,E1 -2541.866,E2 -2541.866} C_VEL
LIN {X 0,Y 566.181,Z 235.456,A -85,B 0,C 180,E1 -2545.024,E2 -2545.024} C_VEL
LIN {X 0,Y 566.162,Z 235.463,A -85,B 0,C 180,E1 -2547.344,E2 -2547.344} C_VEL
LIN {X 0,Y 566.17,Z 235.459,A -85,B 0,C 180,E1 -2549.773,E2 -2549.773} C_VEL
LIN {X 0,Y 566.194,Z 235.452,A -85,B 0,C 180,E1 -2552.43,E2 -2552.43} C_VEL
LIN {X 0,Y 566.168,Z 235.461,A -85,B 0,C 180,E1 -2554.989,E2 -2554.989} C_VEL
LIN {X 0,Y 566.193,Z 235.459,A -85,B 0,C 180,E1 -2557.464,E2 -2557.464} C_VEL
LIN {X 0,Y 566.209,Z 235.452,A -85,B 0,C 180,E1 -2560.201,E2 -2560.201} C_VEL
LIN {X 0,Y 566.182,Z 235.463,A -85,B 0,C 180,E1 -2563.058,E2 -2563.058} C_VEL
LIN {X 0,Y 566.16,Z 235.463,A -85,B 0,C 180,E1 -2566.055,E2 -2566.055} C_VEL
LIN {X 0,Y 566.242,Z 236.037,A -85,B 0,C 180,E1 -2567.081,E2 -2567.081} C_VEL
LIN {X 0,Y 566.574,Z 239.388,A -85,B 0,C 180,E1 -2569.173,E2 -2569.173} C_VEL
LIN {X 0,Y 566.473,Z 243.821,A -85,B 0,C 180,E1 -2571.661,E2 -2571.661} C_VEL
LIN {X 0,Y 566.315,Z 248.762,A -85,B 0,C 180,E1 -2574.32,E2 -2574.32} C_VEL
LIN {X 0,Y 566.275,Z 254.141,A -85,B 0,C 180,E1 -2576.902,E2 -2576.902} C_VEL
LIN {X 0,Y 566.199,Z 259.531,A -85,B 0,C 180,E1 -2579.409,E2 -2579.409} C_VEL
LIN {X 0,Y 566.151,Z 264.92,A -85,B 0,C 180,E1 -2581.855,E2 -2581.855} C_VEL
LIN {X 0,Y 566.11,Z 270.31,A -85,B 0,C 180,E1 -2584.246,E2 -2584.246} C_VEL
LIN {X 0,Y 566.058,Z 276.063,A -85,B 0,C 180,E1 -2586.748,E2 -2586.748} C_VEL
LIN {X 0,Y 566.059,Z 281.089,A -85,B 0,C 180,E1 -2588.897,E2 -2588.897} C_VEL
LIN {X 0,Y 565.985,Z 288.275,A -85,B 0,C 180,E1 -2591.915,E2 -2591.915} C_VEL
LIN {X 0,Y 565.948,Z 295.461,A -85,B 0,C 180,E1 -2594.884,E2 -2594.884} C_VEL
LIN {X 0,Y 565.899,Z 301.524,A -85,B 0,C 180,E1 -2597.357,E2 -2597.357} C_VEL
LIN {X 0,Y 566.911,Z 308.504,A -85,B 0,C 180,E1 -2597.516,E2 -2597.516} C_VEL
LIN {X 0,Y 566.797,Z 321.129,A -85,B 0,C 180,E1 -2597.877,E2 -2597.877} C_VEL
LIN {X 0,Y 566.649,Z 333.465,A -85,B 0,C 180,E1 -2598.373,E2 -2598.373} C_VEL
LIN {X 0,Y 566.539,Z 344.525,A -85,B 0,C 180,E1 -2598.958,E2 -2598.958} C_VEL
LIN {X 0,Y 566.438,Z 355.923,A -85,B 0,C 180,E1 -2599.726,E2 -2599.726} C_VEL
LIN {X 0,Y 566.283,Z 365.583,A -85,B 0,C 180,E1 -2600.535,E2 -2600.535} C_VEL
LIN {X 0,Y 566.175,Z 374.389,A -85,B 0,C 180,E1 -2601.434,E2 -2601.434} C_VEL
LIN {X 0,Y 566.059,Z 383.007,A -85,B 0,C 180,E1 -2602.509,E2 -2602.509} C_VEL
LIN {X 0,Y 565.969,Z 389.872,A -85,B 0,C 180,E1 -2603.583,E2 -2603.583} C_VEL
LIN {X 0,Y 565.937,Z 395.364,A -85,B 0,C 180,E1 -2604.656,E2 -2604.656} C_VEL
LIN {X 0,Y 565.96,Z 399.666,A -85,B 0,C 180,E1 -2605.727,E2 -2605.727} C_VEL
LIN {X 0,Y 565.927,Z 401.964,A -85,B 0,C 180,E1 -2606.44,E2 -2606.44} C_VEL
LIN {X 0,Y 565.878,Z 403.795,A -85,B 0,C 180,E1 -2607.153,E2 -2607.153} C_VEL
LIN {X 0,Y 565.846,Z 406.189,A -85,B 0,C 180,E1 -2608.577,E2 -2608.577} C_VEL
LIN {X 0,Y 565.841,Z 406.782,A -85,B 0,C 180,E1 -2609.288,E2 -2609.288} C_VEL
LIN {X 0,Y 565.841,Z 406.782,A -85,B 0,C 180,E1 -2610.712,E2 -2610.712} C_VEL
LIN {X 0,Y 565.846,Z 406.189,A -85,B 0,C 180,E1 -2611.423,E2 -2611.423} C_VEL
LIN {X 0,Y 565.878,Z 403.795,A -85,B 0,C 180,E1 -2612.847,E2 -2612.847} C_VEL
LIN {X 0,Y 565.927,Z 400.883,A -85,B 0,C 180,E1 -2613.916,E2 -2613.916} C_VEL
LIN {X 0,Y 565.878,Z 396.934,A -85,B 0,C 180,E1 -2614.987,E2 -2614.987} C_VEL
LIN {X 0,Y 565.99,Z 391.84,A -85,B 0,C 180,E1 -2616.059,E2 -2616.059} C_VEL
LIN {X 0,Y 566.035,Z 385.456,A -85,B 0,C 180,E1 -2617.132,E2 -2617.132} C_VEL
LIN {X 0,Y 566.134,Z 377.489,A -85,B 0,C 180,E1 -2618.208,E2 -2618.208} C_VEL
LIN {X 0,Y 566.23,Z 369.348,A -85,B 0,C 180,E1 -2619.105,E2 -2619.105} C_VEL
LIN {X 0,Y 566.336,Z 359.364,A -85,B 0,C 180,E1 -2620.005,E2 -2620.005} C_VEL
LIN {X 0,Y 566.456,Z 349.547,A -85,B 0,C 180,E1 -2620.725,E2 -2620.725} C_VEL
LIN {X 0,Y 566.567,Z 338.77,A -85,B 0,C 180,E1 -2621.366,E2 -2621.366} C_VEL
LIN {X 0,Y 566.731,Z 326.15,A -85,B 0,C 180,E1 -2621.943,E2 -2621.943} C_VEL
LIN {X 0,Y 566.899,Z 313.872,A -85,B 0,C 180,E1 -2622.348,E2 -2622.348} C_VEL
